(* IEC 61131-3 sources: LMM/plc/g, 5 files *)

(* ---- FB_Servo.st ---- *)
FUNCTION_BLOCK FB_Servo
(* =============================================================================
   FB_Servo — 单轴原子封装（SM3_Basic）。仅在 PRG_Axis_Control 任务内实例化。

   仲裁优先级：停止/故障 > 回零 > 绝对定位 > 相对定位 > 速度指令 > 点动。
   - 手动点动走 MC_Jog（松开即减速停）；速度指令走 MC_MoveVelocity
   - 运动切换靠 PLCopen 中止机制（新命令 FB 上升沿自动 abort 旧运动）
   - 全部运动请求撤销（松手/速度归零/停止/急停/撞限位）→ MC_Halt 减速停车
   - 硬限位：xLimEn=TRUE 时，所有模式都限制在 [rLimNeg, rLimPos] 内：
     点动/速度 越限方向被禁止；定位目标被夹紧；X 轴传 xLimEn:=FALSE
   ========================================================================== *)
VAR_IN_OUT
    Axis : AXIS_REF_SM3;
END_VAR
VAR_INPUT
    xEnable : BOOL;         (* 驱动器使能（来自 AxisCmd_xPower） *)
    xStop : BOOL;           (* 停止运动（保持使能） *)
    xResetFault : BOOL;     (* 故障复位（上升沿） *)
    xHome : BOOL;           (* 回零（电平，完成/撤销后由上层清） *)
    xMoveAbs : BOOL;        (* 绝对定位（电平保持至完成） *)
    rTargetPos : REAL;      (* 绝对目标位置 *)
    xMoveRel : BOOL;        (* 相对定位（电平保持至完成） *)
    rDist : REAL;           (* 相对距离（可正可负） *)
    xUseVelCmd : BOOL;      (* 速度指令模式（力跟随/X双驱） *)
    rVelCmd : REAL;         (* 速度给定（可正可负；|v|<1e-6 视为撤销） *)
    xJogPos : BOOL;         (* 点动+（电平，MC_Jog） *)
    xJogNeg : BOOL;         (* 点动-（电平，MC_Jog） *)
    rJogVel : REAL;         (* 点动速度（正值） *)
    rVel : REAL;            (* 定位速度（正值） *)
    rAcc : REAL;            (* 加速度 *)
    rDec : REAL;            (* 减速度 *)
    xLimEn : BOOL;          (* 硬限位使能（X=FALSE，Y/Z/R=TRUE） *)
    rLimPos : REAL;         (* 正方向硬限位（可手动改） *)
    rLimNeg : REAL;         (* 负方向硬限位（可手动改） *)
END_VAR
VAR_OUTPUT
    xPowered : BOOL;        (* 驱动器已上电 := fbPower.Status *)
    xReady : BOOL;          (* 就绪 := 上电且无故障 *)
    xMoving : BOOL;         (* 运动中（含回零） *)
    xStandstill : BOOL;     (* 静止 *)
    xHomed : BOOL;          (* 回零完成（置零后保持） *)
    xFault : BOOL;          (* 故障 := MC_ReadStatus.ErrorStop *)
    xMoveRelDone : BOOL;    (* 相对定位完成 *)
    xMoveAbsDone : BOOL;    (* 绝对定位完成 *)
    rActPos : LREAL;        (* 实际位置 *)
    (* --- 诊断输出（g 线 0.5 新增；上层可不接线，在线直接看） --- *)
    xVelReq : BOOL;         (* 诊断：仲裁后速度请求已成立 *)
    xVelBusy : BOOL;        (* 诊断：MC_MoveVelocity.Busy *)
    xVelInVel : BOOL;       (* 诊断：MC_MoveVelocity.InVelocity *)
    xErrPower : BOOL;       (* 诊断：MC_Power.Error（驱动未就绪/通讯异常） *)
    xErrVel : BOOL;         (* 诊断：MC_MoveVelocity.Error（参数/平台拒绝） *)
    xErrJog : BOOL;         (* 诊断：MC_Jog.Error *)
    xErrHalt : BOOL;        (* 诊断：MC_Halt.Error *)
    xErrHome : BOOL;        (* 诊断：MC_Home.Error *)
    xErrAbs : BOOL;         (* 诊断：MC_MoveAbsolute.Error *)
    xErrRel : BOOL;         (* 诊断：MC_MoveRelative.Error *)
END_VAR
VAR
    fbPower : MC_Power;
    fbHalt : MC_Halt;
    fbHome : MC_Home;
    fbReset : MC_Reset;
    fbReadStatus : MC_ReadStatus;
    fbReadPos : MC_ReadActualPosition;
    fbSetPos : MC_SetPosition;
    fbMoveRel : MC_MoveRelative;
    fbMoveAbs : MC_MoveAbsolute;
    fbMoveVel : MC_MoveVelocity;
    fbJog : MC_Jog;
    eDir : MC_DIRECTION;
    xReqStop : BOOL;
    xReqHome : BOOL;
    xReqAbs : BOOL;
    xReqRel : BOOL;
    xReqVel : BOOL;
    xReqJogPos : BOOL;
    xReqJogNeg : BOOL;
    xReqAny : BOOL;
    xReqHomePrev : BOOL;
    xSetZeroTrig : BOOL;
    xVelRunPrev : BOOL;
    xDirFlip : BOOL;
    xNeedStop : BOOL;
    xHaltPrev : BOOL;
    xResetPrev : BOOL;
    xBlockPos : BOOL;
    xBlockNeg : BOOL;
    rAbsTarget : REAL;
    rRelDist : REAL;
    rVelInPrev : REAL;
END_VAR

(* 1. 状态与位置 *)
fbReadStatus(Axis := Axis, Enable := TRUE);
fbReadPos(Axis := Axis, Enable := TRUE);
rActPos := fbReadPos.Position;
xStandstill := fbReadStatus.StandStill;
xFault := fbReadStatus.ErrorStop;
xMoving := fbReadStatus.DiscreteMotion OR fbReadStatus.ContinuousMotion OR fbReadStatus.Homing;

(* 2. 故障复位（上升沿） *)
fbReset(Axis := Axis, Execute := xResetFault AND NOT xResetPrev);
xResetPrev := xResetFault;

(* 3. 驱动器使能（xStop 不掉使能） *)
fbPower(Axis := Axis, Enable := TRUE,
        bRegulatorOn := xEnable AND NOT xFault,
        bDriveStart := xEnable AND NOT xFault);
xPowered := fbPower.Status;
xReady := xPowered AND NOT xFault;

(* 4. 硬限位：越限方向禁止；定位目标夹紧（已越限时仍允许向回运动） *)
xBlockPos := xLimEn AND (rActPos >= rLimPos);
xBlockNeg := xLimEn AND (rActPos <= rLimNeg);
rAbsTarget := rTargetPos;
rRelDist := rDist;
IF xLimEn THEN
    rAbsTarget := LIMIT(rLimNeg, rTargetPos, rLimPos);
    rRelDist := LIMIT(rLimNeg, rActPos + rDist, rLimPos) - rActPos;
END_IF;

(* 5. 命令仲裁：停止/故障 > 回零 > 绝对 > 相对 > 速度 > 点动 *)
xReqStop := xStop OR NOT xEnable OR xFault;
xReqHome := xHome AND NOT xReqStop;
xReqAbs := xMoveAbs AND xPowered AND NOT xReqStop AND NOT xReqHome;
xReqRel := xMoveRel AND (ABS(rRelDist) > 1.0E-9) AND xPowered
           AND NOT xReqStop AND NOT xReqHome AND NOT xReqAbs;
xReqVel := xUseVelCmd AND (ABS(rVelCmd) > 1.0E-6) AND xPowered
           AND NOT ((rVelCmd > 0.0) AND xBlockPos) AND NOT ((rVelCmd < 0.0) AND xBlockNeg)
           AND NOT xReqStop AND NOT xReqHome AND NOT xReqAbs AND NOT xReqRel;
xReqJogPos := xJogPos AND NOT xJogNeg AND NOT xBlockPos AND xPowered
              AND NOT xReqStop AND NOT xReqHome AND NOT xReqAbs AND NOT xReqRel AND NOT xReqVel;
xReqJogNeg := xJogNeg AND NOT xJogPos AND NOT xBlockNeg AND xPowered
              AND NOT xReqStop AND NOT xReqHome AND NOT xReqAbs AND NOT xReqRel AND NOT xReqVel;
xReqAny := xReqHome OR xReqAbs OR xReqRel OR xReqVel OR xReqJogPos OR xReqJogNeg;

(* 6. 回零：MC_Home(0) → MC_SetPosition(0) → xHomed *)
IF xReqHome AND NOT xReqHomePrev THEN
    xHomed := FALSE;
END_IF;
xReqHomePrev := xReqHome;
fbHome(Axis := Axis, Execute := xReqHome, Position := 0.0);
IF fbHome.Done THEN
    xSetZeroTrig := TRUE;
END_IF;
fbSetPos(Axis := Axis, Execute := xSetZeroTrig, Position := 0.0);
IF fbSetPos.Done THEN
    xHomed := TRUE;
    xSetZeroTrig := FALSE;
END_IF;

(* 7. 绝对 / 相对定位（目标已夹紧；电平保持 Execute，Done 上报） *)
fbMoveAbs(Axis := Axis, Execute := xReqAbs, Position := rAbsTarget,
          Velocity := ABS(rVel), Acceleration := rAcc, Deceleration := rDec);
fbMoveRel(Axis := Axis, Execute := xReqRel, Distance := rRelDist,
          Velocity := ABS(rVel), Acceleration := rAcc, Deceleration := rDec);
xMoveAbsDone := fbMoveAbs.Done;
xMoveRelDone := fbMoveRel.Done;

(* 8. 速度指令：MC_MoveVelocity；Velocity 取绝对值，方向走 Direction *)
(* 注意：本机 SM3 库的方向字面值是 positive/negative（非 CoDeSys 的 mcPositiveDirection） *)
IF rVelCmd >= 0.0 THEN
    eDir := positive;
ELSE
    eDir := negative;
END_IF;
(* 运行中换向：先撤 Execute 一拍，下一拍带新方向重新触发 *)
xDirFlip := xReqVel AND xVelRunPrev AND ((rVelCmd >= 0.0) <> (rVelInPrev >= 0.0));
fbMoveVel(Axis := Axis, Execute := xReqVel AND NOT xDirFlip,
          Velocity := ABS(rVelCmd), Direction := eDir,
          Acceleration := rAcc, Deceleration := rDec);
xVelRunPrev := xReqVel;
rVelInPrev := rVelCmd;

(* 9. 手动点动：MC_Jog（按住动、松开减速停；越限方向已在仲裁禁止） *)
fbJog(Axis := Axis,
      JogForward := xReqJogPos,
      JogBackward := xReqJogNeg,
      Velocity := ABS(rJogVel),
      Acceleration := rAcc,
      Deceleration := rDec);

(* 10. 停车：有使能但无任何运动请求（松手/速度归零/停止/急停/撞限位）→ MC_Halt *)
xNeedStop := xPowered AND NOT xReqAny;
fbHalt(Axis := Axis, Execute := xNeedStop AND xMoving AND NOT xHaltPrev,
       Deceleration := rDec);
xHaltPrev := xNeedStop AND xMoving;

(* 11. 诊断输出（g 线 0.5） *)
xVelReq := xReqVel;
xVelBusy := fbMoveVel.Busy;
xVelInVel := fbMoveVel.InVelocity;
xErrPower := fbPower.Error;
xErrVel := fbMoveVel.Error;
xErrJog := fbJog.Error;
xErrHalt := fbHalt.Error;
xErrHome := fbHome.Error;
xErrAbs := fbMoveAbs.Error;
xErrRel := fbMoveRel.Error;

(* ---- FB_XDual.st ---- *)
FUNCTION_BLOCK FB_XDual
(* ==============================================================================
 * FB_XDual — X 轴双驱（g 线 0.59）：单沿起步 + SM3 斜坡 + Halt 对称减速
 * 铁律：X 轴只经本 FB；FB_Servo 不得持有 X 轴实例。
 *
 *   0.44 根因：Enable 和调节器一起关 → Power FB 停转，驱动收不到卸使能；
 *   运动中切使能 + 刚上使能就 Execute → 连冲、Error 锁死第二次点动。
 *   对齐 FB_Servo：Enable 保持，bRegulatorOn/bDriveStart 跟 xRegOn；
 *   松手 Halt 脉冲刹停，双轴 standstill 后才卸调节器；2s 未静止改发 Stop。
 *   冷启动等 Status 约 80ms 且双轴 standstill 再出速度；短窗内再按不再等。
 *   0.47：禁止 300ms 超时在减速中卸使能（运动中送掉使能报错）。
 *   0.50：幅值差速不撤 Execute。必须重触发的只有换向。
 *   0.51：0.50 仍三次过冲——使能后 20ms 就 Execute（失败连打）+ 爬坡每拍改 Velocity。
 *         上使能后等 Status 80ms；Error 锁 150ms；爬坡只吃基速，到速后再跟 trim。
 *   0.52：xErrVel 不跳仍冲三次+忽快忽慢。根因是 0.51 把 xPowerSettled 绑在 standstill：
 *         轴一动就掉 Execute，松手前 Acc/Dec 反复爬。闭锁一次后保持；残差 P 降增益。
 *   0.53：xVelReq 一直 TRUE 仍冲三次。请求≠Execute；Acc=Jog 时 SM3 梯形拐点 + 使能冲击叠成三次。
 *         PLC 按用户 Acc 爬 FB 速度，SM3 Acc 抬到 ≥10 只负责跟上；松手仍 Halt。
 *   0.54：0.53 不过冲也不走。本机 Execute 保持时 Velocity 不刷新，第一拍 ~0 被锁死。
 *         上升沿一次写入目标速度 + 用户 Acc；爬坡中不改输入；到速后再跟 trim。
 *   0.55：三次过冲=Execute 被拉了三次。PRG_Logic 先清 AxisCmd 再置位，ETHERCAT(prio0)
 *         在 FALSE 空窗采到松手→Halt→再加速。第一次点动 Logic 超时约 3 拍。去抖+一次写入。
 *   0.56：偶发三次过冲。0.55 去抖保了 eMode，但 Power.Status 闪一下仍清 xStartReady，
 *         Execute 掉、锁存清 0，再启动就是又一次过冲。点动中 Execute 闭锁到松开。
 *   0.57：现场仍每次起步沿 X 往复冲 3 次（约 3s）。根因：起步=速度阶跃（Acc=25）
 *         打进 CSV 速度环，激起双驱耦合龙门 ~1Hz 纵向共振。0.53 阶梯爬速本可消过冲，
 *         但本机 Execute 保持时 Velocity 不刷新，首拍 ~0 锁死（"不过冲也不走"）。
 *   0.58：恢复 rVelSlew 阶梯爬速；爬坡期 Execute 每步重触发（OFF/ON 交替一拍，
 *         上升沿重采样）；斜率取用户 Acc/Dec 钳 [0.05, rRampAccMax]，SM3 Acc 只跟梯；
 *         松手/到位先阶梯降到 ~0 再 Halt；MoveRel 剩余≤slew²/2Dec 提前减速；
 *         到位锁 xDecelDone 禁停稳后重爬目标。
 *   0.59：0.58 每步重触发 = 250Hz 沿风暴，现场 acc=0.8 起步仍快速冲 2 次（~1s）、
 *         第三次慢、停死；M2 明显慢于 M1（两侧接受沿时刻不一致，M2 漏沿爬速落后）。
 *         改单沿起步：一个上升沿写最终目标 + 钳制用户 Acc/Dec（0.05~1.0），
 *         SM3 自带斜坡 0→目标（0.8 → 0.5s）；稳态 trim/sync 更新走限频重触发
 *         （≥200ms 一次、差值≥0.004）；减速统一 Halt（用户 Dec 对称）。
 * ============================================================================== *)
VAR_IN_OUT
    AxisM1 : AXIS_REF_SM3;
    AxisM2 : AXIS_REF_SM3;
END_VAR
VAR_INPUT
    xEnable : BOOL;
    xStop : BOOL;
    xResetFault : BOOL;
    xJogPos : BOOL;
    xJogNeg : BOOL;
    xSpinLeft : BOOL;
    xSpinRight : BOOL;
    xMoveRel : BOOL;
    rMoveDist : REAL;
    rMoveVel : REAL;
    rJogVel : REAL;
    rSpinVel : REAL;
    rHeadingErr : REAL;
    rKpTrack : REAL;
    rAcc : REAL;
    rDec : REAL;
    rTrimMax : REAL;
    xSyncEnable : BOOL := TRUE;
    rRatioM1 : REAL := 1.0;
    rRatioM2 : REAL := 1.0;
    rHeadingDeadband : REAL := 0.003;
    rTrimFilterTc : REAL := 0.05;
    rCycleSec : REAL := 0.004;
    (* 0.60 外部直控（视觉直写 M1/M2 速度）：xDirectMode=TRUE 时绕过 trim/sync *)
    xDirectMode : BOOL;
    rVelM1Direct : REAL;
    rVelM2Direct : REAL;
    tDirectRetrig : TIME := T#40MS;
END_VAR
VAR_OUTPUT
    xMoveDone : BOOL;
    rPosV : REAL;
    rSyncErr : REAL;
    rVelFactor : REAL;
    xCoupled : BOOL;
    xInGearM1 : BOOL;
    xInGearM2 : BOOL;
    xPoweredV : BOOL;
    xSyncWarn : BOOL;
    xSyncFault : BOOL;
    iState : INT;
    iHoldState : INT;
    eSlaveMode : INT;
    rVelCmdM1 : REAL;
    rVelCmdM2 : REAL;
    rPosM1 : REAL;
    rPosM2 : REAL;
    xMovingM1 : BOOL;
    xMovingM2 : BOOL;
    xStandstillM1 : BOOL;
    xStandstillM2 : BOOL;
    xPoweredM1 : BOOL;
    xPoweredM2 : BOOL;
    xReadyM1 : BOOL;
    xReadyM2 : BOOL;
    xFaultM1 : BOOL;
    xFaultM2 : BOOL;
    xVelReqM1 : BOOL;
    xVelReqM2 : BOOL;
    xVelBusyM1 : BOOL;
    xVelBusyM2 : BOOL;
    xErrPowerM1 : BOOL;
    xErrPowerM2 : BOOL;
    xErrVelM1 : BOOL;
    xErrVelM2 : BOOL;
    xVelExecM1 : BOOL;
    xVelExecM2 : BOOL;
    xVelInVelM1 : BOOL;
    xVelInVelM2 : BOOL;
    iVelExecRise : INT;
    rVelActM1Out : REAL;
    rVelActM2Out : REAL;
    xDirectActive : BOOL;
END_VAR
VAR
    fbPowerM1 : MC_Power;
    fbPowerM2 : MC_Power;
    fbResetM1 : MC_Reset;
    fbResetM2 : MC_Reset;
    fbVelM1 : MC_MoveVelocity;
    fbVelM2 : MC_MoveVelocity;
    fbHaltM1 : MC_Halt;
    fbHaltM2 : MC_Halt;
    fbStopM1 : MC_Stop;
    fbStopM2 : MC_Stop;
    eDirM1 : MC_DIRECTION;
    eDirM2 : MC_DIRECTION;
    eMode : INT;
    eModePrev : INT;
    rBase : REAL;
    rVelActM1 : REAL;
    rVelActM2 : REAL;
    rTrim : REAL;
    rTrimRaw : REAL;
    rTrimFiltered : REAL;
    rAlphaFilter : REAL;
    rUseRatioM1 : REAL;
    rUseRatioM2 : REAL;
    rSyncExpect : REAL;
    rSyncResid : REAL;
    rCorrPos : REAL;
    rCorrV1 : REAL;
    rCorrV2 : REAL;
    rVelFF1 : REAL;
    rVelFF2 : REAL;
    rKpSync : REAL := 0.05;
    rKvSync : REAL := 0.0;
    rSyncDeadband : REAL := 0.02;
    rCorrPosMax : REAL := 0.08;
    rCorrVelMax : REAL := 0.06;
    xStraightEdge : BOOL;
    xJogRaw : BOOL;
    xJogHeld : BOOL;
    tonJogOff : TON;
    tonStillM1 : TON;
    tonStillM2 : TON;
    tonHoldFallback : TON;
    tonJogGrace : TON;
    rHoldVelMax : REAL := 0.5;
    xSoftHold : BOOL;
    xSoftHoldPrev : BOOL;
    xSoftHoldLatched : BOOL;
    fbSetPosM1 : MC_SetPosition;
    fbSetPosM2 : MC_SetPosition;
    xZeroGate : BOOL;
    tonZeroDelay : TON;
    xZeroReady : BOOL;
    xZeroPulsePrev : BOOL;
    xSetPosReq : BOOL;
    xPosZeroed : BOOL;
    xErrSetPosM1 : BOOL;
    xErrSetPosM2 : BOOL;
    xResetEdge : BOOL;
    xResetPrev : BOOL;
    xDirFlipM1 : BOOL;
    xDirFlipM2 : BOOL;
    xVelRunPrevM1 : BOOL;
    xVelRunPrevM2 : BOOL;
    rVelInPrevM1 : REAL;
    rVelInPrevM2 : REAL;
    rVelAppl : REAL;
    rAccUse : REAL;
    rDecUse : REAL;
    rAccLatch : REAL;
    rDecLatch : REAL;
    rVelLatchM1 : REAL;
    rVelLatchM2 : REAL;
    xExecPrev : BOOL;
    rAccSoftMin : REAL := 0.05;
    rAccSoft : REAL;
    rDecSoft : REAL;
    rRampAccMax : REAL := 1.0;
    xDecelActive : BOOL;
    xDecelDone : BOOL;
    rDecelDist : REAL;
    xM1Decel : BOOL;
    xM2Decel : BOOL;
    xBothPowered : BOOL;
    xPowerGate : BOOL;
    xReqVelM1 : BOOL;
    xReqVelM2 : BOOL;
    xNeedHaltM1 : BOOL;
    xNeedHaltM2 : BOOL;
    xRegOn : BOOL;
    xRegOnPrev : BOOL;
    xStopping : BOOL;
    xWasStopping : BOOL;
    xHaltTrig : BOOL;
    xHaltPrev : BOOL;
    xPowerSettled : BOOL;
    xStartReady : BOOL;
    xStopFallback : BOOL;
    tonHaltWin : TON;
    tonPowerOk : TON;
    tonVelHold : TON;
    tonRampLock : TON;
    tonTrimRetrig : TON;
    xTrimWant : BOOL;
    xTrimPulse : BOOL;
    xTrimPulsePrev : BOOL;
    xMoveRelDecelTrig : BOOL;
    xExecM1 : BOOL;
    xExecHold : BOOL;
    xHaltBusy : BOOL;
    xExecBoth : BOOL;
    xDirFlipAny : BOOL;
    xVelHoldOff : BOOL;
    xErrVelPrev : BOOL;
    xRampLock : BOOL;
    rVelFbM1 : REAL;
    rVelFbM2 : REAL;
    rVelFbHoldM1 : REAL;
    rVelFbHoldM2 : REAL;
    rCorrLim : REAL;
    xMovePrev : BOOL;
    xArmed : BOOL;
    rStart : REAL;
    rAvg : REAL;
    rSyncWarnLevel : REAL := 0.05;
    rSyncFaultLevel : REAL := 0.15;
    tonSyncFault : TON;
    tonDirectRetrig : TON;
    xDirectWant : BOOL;
    xDirectPulse : BOOL;
    xDirectPulsePrev : BOOL;
    xHaltDemand : BOOL;
END_VAR

rVelFactor := 0.0;
xCoupled := FALSE;
xInGearM1 := FALSE;
xInGearM2 := FALSE;
xPoweredV := FALSE;
eSlaveMode := 0;

(* ------------------- 1. 模式 ------------------- *)
(* 点动 FALSE 短于 40ms 视为空窗，不 Halt、不撤 Execute *)
xJogRaw := (xJogPos XOR xJogNeg) OR xMoveRel;
tonJogOff(IN := xJogHeld AND NOT xJogRaw AND xEnable AND NOT xStop
           AND NOT (xSpinLeft XOR xSpinRight), PT := T#40MS);
IF xStop OR NOT xEnable THEN
    eMode := 0;
    rBase := 0.0;
    xJogHeld := FALSE;
ELSIF xSpinLeft XOR xSpinRight THEN
    IF xSpinLeft THEN
        eMode := 2;
    ELSE
        eMode := 3;
    END_IF;
    rBase := 0.0;
    xJogHeld := FALSE;
ELSIF xDirectMode THEN
    (* 0.60 外部直控优先于点动：视觉接管期间忽略点动/走距输入 *)
    eMode := 4;
    rBase := 0.0;
    xJogHeld := FALSE;
ELSIF xJogRaw THEN
    eMode := 1;
    xJogHeld := TRUE;
    IF xMoveRel THEN
        IF rMoveDist >= 0.0 THEN
            rBase := ABS(rMoveVel);
        ELSE
            rBase := -ABS(rMoveVel);
        END_IF;
    ELSIF xJogPos THEN
        rBase := ABS(rJogVel);
    ELSE
        rBase := -ABS(rJogVel);
    END_IF;
ELSIF xJogHeld AND NOT tonJogOff.Q THEN
    eMode := 1;
ELSE
    eMode := 0;
    rBase := 0.0;
    xJogHeld := FALSE;
END_IF;
iState := eMode;
xStraightEdge := (eMode = 1) AND (eModePrev <> 1);

(* ------------------- 2. 回读 + SoftHold ------------------- *)
rPosM1 := LREAL_TO_REAL(AxisM1.fActPosition);
rPosM2 := LREAL_TO_REAL(AxisM2.fActPosition);
rVelActM1 := LREAL_TO_REAL(AxisM1.fActVelocity);
rVelActM2 := LREAL_TO_REAL(AxisM2.fActVelocity);
rAvg := (rPosM1 + rPosM2) * 0.5;
rPosV := rAvg;
rSyncErr := rPosM1 - rPosM2;

xStandstillM1 := AxisM1.nAxisState = SMC_AXIS_STATE.standstill;
xStandstillM2 := AxisM2.nAxisState = SMC_AXIS_STATE.standstill;
xMovingM1 := (NOT xStandstillM1) OR (ABS(rVelActM1) > 0.01);
xMovingM2 := (NOT xStandstillM2) OR (ABS(rVelActM2) > 0.01);

tonStillM1(IN := NOT xMovingM1, PT := T#200MS);
tonStillM2(IN := NOT xMovingM2, PT := T#200MS);
tonHoldFallback(IN := (eMode = 0) AND NOT xStop AND xEnable
                    AND (ABS(rVelActM1) < rHoldVelMax) AND (ABS(rVelActM2) < rHoldVelMax),
                PT := T#2S);
IF xStop OR NOT xEnable OR (eMode <> 0) THEN
    iHoldState := 0;
    xSoftHoldLatched := FALSE;
ELSIF xSoftHoldLatched THEN
    iHoldState := 2;
ELSIF (tonStillM1.Q AND tonStillM2.Q) OR tonHoldFallback.Q THEN
    iHoldState := 2;
    xSoftHoldLatched := TRUE;
ELSE
    iHoldState := 1;
END_IF;
xSoftHold := iHoldState = 2;
xSoftHoldPrev := xSoftHold;
(* 再按起步 300ms 内隐藏 SoftHold/Halt 残留 bError，避免 Fault→StopAll 发肉 *)
tonJogGrace(IN := (eMode <> 0), PT := T#300MS);

xSyncWarn := ABS(rSyncErr) > rSyncWarnLevel;
tonSyncFault(IN := ABS(rSyncErr) > rSyncFaultLevel, PT := T#500MS);
IF tonSyncFault.Q THEN
    xSyncFault := TRUE;
END_IF;

(* ------------------- 3. 复位仅手动 ------------------- *)
fbResetM1(Axis := AxisM1, Execute := xResetFault);
fbResetM2(Axis := AxisM2, Execute := xResetFault);
IF xResetFault THEN
    xSyncFault := FALSE;
END_IF;

(* ------------------- 4. 使能：Power.Enable 常开，只切调节器 ------------------- *)
(* 松手保持调节器直到双轴 standstill。300ms 超时会在减速未完时卸使能（0.46 报错）。 *)
xWasStopping := xStopping;
IF xStop OR NOT xEnable THEN
    xStopping := FALSE;
ELSIF eMode <> 0 THEN
    xStopping := FALSE;
ELSIF xRegOnPrev THEN
    xStopping := TRUE;
END_IF;
tonHaltWin(IN := xStopping AND (eMode = 0) AND xEnable AND NOT xStop, PT := T#2S);
IF xStopping AND (eMode = 0) AND xStandstillM1 AND xStandstillM2 THEN
    xStopping := FALSE;
END_IF;
xRegOn := xEnable AND NOT xStop AND ((eMode <> 0) OR xStopping);
xStopFallback := xStopping AND tonHaltWin.Q AND NOT (xStandstillM1 AND xStandstillM2) AND NOT xDecelActive;
(* Enable 恒 TRUE，卸使能只走调节器（对齐 FB_Servo；0.44 关 Enable 导致驱动收不到） *)
fbPowerM1(Axis := AxisM1, Enable := TRUE,
          bRegulatorOn := xRegOn, bDriveStart := xRegOn);
fbPowerM2(Axis := AxisM2, Enable := TRUE,
          bRegulatorOn := xRegOn, bDriveStart := xRegOn);

xPoweredM1 := fbPowerM1.Status;
xPoweredM2 := fbPowerM2.Status;
xFaultM1 := AxisM1.bError AND xRegOn AND NOT (xSoftHold OR (iHoldState = 1) OR xStopping OR ((eMode <> 0) AND NOT tonJogGrace.Q));
xFaultM2 := AxisM2.bError AND xRegOn AND NOT (xSoftHold OR (iHoldState = 1) OR xStopping OR ((eMode <> 0) AND NOT tonJogGrace.Q));
(* 故意停调节器时仍报就绪，避免 Logic 1007 *)
xReadyM1 := xEnable AND NOT xStop AND NOT xFaultM1;
xReadyM2 := xEnable AND NOT xStop AND NOT xFaultM2;
xBothPowered := xPoweredM1 AND xPoweredM2;
xPowerGate := xEnable AND NOT xStop AND NOT xFaultM1 AND NOT xFaultM2;
tonPowerOk(IN := xRegOn AND xBothPowered AND (eMode <> 0), PT := T#80MS);
(* 冷启动闭锁一次。Status 闪烁不得清 xStartReady，否则 Execute 掉了再爬。 *)
IF (eMode = 0) OR NOT xRegOn OR xStop THEN
    xStartReady := FALSE;
ELSIF xWasStopping OR xExecHold THEN
    xStartReady := TRUE;
ELSIF tonPowerOk.Q AND xStandstillM1 AND xStandstillM2 THEN
    xStartReady := TRUE;
END_IF;
xPowerSettled := xRegOn AND (eMode <> 0) AND xStartReady
                 AND (xBothPowered OR xExecHold);

(* 置零：点动/短窗禁止；空闲自动置零会和 Halt 抢轴，只保留手动 Reset *)
IF (eMode <> 0) OR xStopping OR xStop OR NOT xEnable THEN
    xSetPosReq := FALSE;
END_IF;
xZeroGate := FALSE;
tonZeroDelay(IN := FALSE, PT := T#300MS);
xZeroReady := FALSE;
xZeroPulsePrev := FALSE;
xResetEdge := xResetFault AND NOT xResetPrev;
xResetPrev := xResetFault;
IF xResetEdge AND (eMode = 0) AND NOT xStopping THEN
    xSetPosReq := TRUE;
END_IF;
fbSetPosM1(Axis := AxisM1, Execute := xSetPosReq AND (eMode = 0) AND NOT xStopping, Position := 0.0);
fbSetPosM2(Axis := AxisM2, Execute := xSetPosReq AND (eMode = 0) AND NOT xStopping, Position := 0.0);
xErrSetPosM1 := fbSetPosM1.Error;
xErrSetPosM2 := fbSetPosM2.Error;
IF xSetPosReq THEN
    IF (fbSetPosM1.Done AND fbSetPosM2.Done) OR fbSetPosM1.Error OR fbSetPosM2.Error THEN
        xSetPosReq := FALSE;
        xPosZeroed := TRUE;
    END_IF;
END_IF;

(* ------------------- 6. 基速跟手 + 视觉差速 ------------------- *)
rAccUse := ABS(rAcc);
IF rAccUse < rAccSoftMin THEN
    rAccUse := rAccSoftMin;
END_IF;
rDecUse := ABS(rDec);
IF rDecUse < rAccSoftMin THEN
    rDecUse := rAccSoftMin;
END_IF;

(* 0.59：SM3 斜坡用钳制 Acc/Dec（0.05~rRampAccMax）。HMI 25/100 兜底不再变阶跃；
   rDecUse 保留软下限继续供 Stop 急停。 *)
rAccSoft := ABS(rAcc);
IF rAccSoft < rAccSoftMin THEN
    rAccSoft := rAccSoftMin;
END_IF;
IF rAccSoft > rRampAccMax THEN
    rAccSoft := rRampAccMax;
END_IF;
rDecSoft := ABS(rDec);
IF rDecSoft < rAccSoftMin THEN
    rDecSoft := rAccSoftMin;
END_IF;
IF rDecSoft > rRampAccMax THEN
    rDecSoft := rRampAccMax;
END_IF;

(* 0.36：禁止 PLC 再爬 rVelAppl。按下即目标速度，松开即 0，停靠 Halt。 *)
(* 0.59 注：rVelAppl 是最终目标；起步斜坡由 SM3 按 rAccSoft 生成（单沿锁存）。 *)
IF (eMode = 0) OR xStop OR NOT xEnable THEN
    rVelAppl := 0.0;
ELSIF eMode = 1 THEN
    rVelAppl := rBase;
ELSE
    rVelAppl := 0.0;
END_IF;

(* 视觉：同一条基速上 ±trim，不是第二次运动，不撤 Execute *)
rTrimRaw := 0.0;
rCorrPos := 0.0;
rCorrV1 := 0.0;
rCorrV2 := 0.0;
rUseRatioM1 := rRatioM1;
IF rUseRatioM1 < 0.1 THEN
    rUseRatioM1 := 0.1;
END_IF;
rUseRatioM2 := rRatioM2;
IF rUseRatioM2 < 0.1 THEN
    rUseRatioM2 := 0.1;
END_IF;
IF eMode = 1 THEN
    IF ABS(rHeadingErr) > ABS(rHeadingDeadband) THEN
        IF rHeadingErr > 0.0 THEN
            rTrimRaw := (rHeadingErr - ABS(rHeadingDeadband)) * rKpTrack;
        ELSE
            rTrimRaw := (rHeadingErr + ABS(rHeadingDeadband)) * rKpTrack;
        END_IF;
        rTrimRaw := LIMIT(-ABS(rTrimMax), rTrimRaw, ABS(rTrimMax));
    END_IF;
    IF rTrimFilterTc > 0.001 THEN
        rAlphaFilter := rCycleSec / (rTrimFilterTc + rCycleSec);
        rTrimFiltered := rTrimFiltered + rAlphaFilter * (rTrimRaw - rTrimFiltered);
    ELSE
        rTrimFiltered := rTrimRaw;
    END_IF;
    rTrim := rTrimFiltered;
    IF xStraightEdge THEN
        rSyncExpect := rPosM1 - rPosM2;
        rTrimFiltered := 0.0;
        rTrim := 0.0;
        xRampLock := TRUE;
    END_IF;
    rSyncExpect := rSyncExpect + (2.0 * rTrim * rCycleSec);
    rSyncResid := (rPosM1 - rPosM2) - rSyncExpect;
    rCorrLim := ABS(rCorrPosMax);
    IF ABS(rVelAppl) > 0.001 THEN
        IF (0.25 * ABS(rVelAppl)) < rCorrLim THEN
            rCorrLim := 0.25 * ABS(rVelAppl);
        END_IF;
    END_IF;
    IF xSyncEnable AND (ABS(rVelAppl) > 0.001) THEN
        IF ABS(rSyncResid) > rSyncDeadband THEN
            rCorrPos := LIMIT(-rCorrLim, rKpSync * rSyncResid, rCorrLim);
        END_IF;
        rCorrV1 := LIMIT(-ABS(rCorrVelMax), rKvSync * ((rVelAppl + rTrim) - rVelActM1), ABS(rCorrVelMax));
        rCorrV2 := LIMIT(-ABS(rCorrVelMax), rKvSync * ((rVelAppl - rTrim) - rVelActM2), ABS(rCorrVelMax));
    END_IF;
    rVelFF1 := rVelAppl + rTrim;
    rVelFF2 := rVelAppl - rTrim;
    rVelCmdM1 := (rVelFF1 - 0.5 * rCorrPos + rCorrV1) * rUseRatioM1;
    rVelCmdM2 := (rVelFF2 + 0.5 * rCorrPos + rCorrV2) * rUseRatioM2;
    IF ABS(rVelAppl) > 0.001 THEN
        IF rVelAppl > 0.0 THEN
            IF rVelCmdM1 < 0.0 THEN
                rVelCmdM1 := 0.0;
            END_IF;
            IF rVelCmdM2 < 0.0 THEN
                rVelCmdM2 := 0.0;
            END_IF;
        ELSE
            IF rVelCmdM1 > 0.0 THEN
                rVelCmdM1 := 0.0;
            END_IF;
            IF rVelCmdM2 > 0.0 THEN
                rVelCmdM2 := 0.0;
            END_IF;
        END_IF;
    END_IF;
ELSIF (eMode = 2) OR (eMode = 3) THEN
    rTrimFiltered := 0.0;
    IF eMode = 2 THEN
        rVelCmdM1 := ABS(rSpinVel) * rUseRatioM1;
    ELSE
        rVelCmdM1 := -ABS(rSpinVel) * rUseRatioM1;
    END_IF;
    rVelCmdM2 := -rVelCmdM1 * (rUseRatioM2 / rUseRatioM1);
ELSIF eMode = 4 THEN
    (* 0.60 外部直控：两个速度直接来自视觉，不做 trim/sync/斜坡 *)
    rTrimFiltered := 0.0;
    rVelCmdM1 := rVelM1Direct * rUseRatioM1;
    rVelCmdM2 := rVelM2Direct * rUseRatioM2;
ELSE
    rTrimFiltered := 0.0;
    rVelCmdM1 := rVelAppl;
    rVelCmdM2 := rVelAppl;
END_IF;
IF xStop OR NOT xEnable THEN
    rVelCmdM1 := 0.0;
    rVelCmdM2 := 0.0;
END_IF;
IF eMode <> 1 THEN
    xRampLock := FALSE;
ELSIF xRampLock THEN
    IF (ABS(rVelAppl) > 0.001)
            AND (ABS(rVelActM1) >= 0.8 * ABS(rVelAppl))
            AND (ABS(rVelActM2) >= 0.8 * ABS(rVelAppl)) THEN
        xRampLock := FALSE;
    END_IF;
END_IF;
tonRampLock(IN := xRampLock AND (eMode = 1), PT := T#800MS);
IF tonRampLock.Q THEN
    xRampLock := FALSE;
END_IF;
IF (eMode = 1) AND xRampLock THEN
    rVelFbM1 := rVelAppl * rUseRatioM1;
    rVelFbM2 := rVelAppl * rUseRatioM2;
ELSE
    rVelFbM1 := rVelCmdM1;
    rVelFbM2 := rVelCmdM2;
END_IF;
IF (eMode <> 1) OR xStraightEdge THEN
    rVelFbHoldM1 := rVelFbM1;
    rVelFbHoldM2 := rVelFbM2;
ELSE
    IF ABS(rVelFbM1 - rVelFbHoldM1) < 0.004 THEN
        rVelFbM1 := rVelFbHoldM1;
    ELSE
        rVelFbHoldM1 := rVelFbM1;
    END_IF;
    IF ABS(rVelFbM2 - rVelFbHoldM2) < 0.004 THEN
        rVelFbM2 := rVelFbHoldM2;
    ELSE
        rVelFbHoldM2 := rVelFbM2;
    END_IF;
END_IF;

(* ------------------- 7. 双轴 MoveVelocity ------------------- *)
(* 0.54：上升沿锁目标。0.58 每步重触发被 0.59 废除：250Hz 沿风暴反复踢起龙门
   1Hz 共振（现场 acc=0.8：起步快速冲 2 次 ~1s、第三次慢、停死）；两侧 FB/驱动
   接受沿时刻不一致 → M2 漏沿爬速落后（M2 明显慢）。0.59：起步只发一个上升沿，
   一次写入最终目标 + 钳制 Acc/Dec，SM3 自带斜坡 0→目标（0.8 → 0.5s）；
   稳态 trim/sync 更新走限频重触发；减速由 Halt 接管（见第 8 节）。 *)
xHaltBusy := fbHaltM1.Busy OR fbHaltM2.Busy OR fbStopM1.Busy OR fbStopM2.Busy;
IF (eMode = 1) AND xPowerGate AND xPowerSettled AND (ABS(rVelAppl) > 0.001)
        AND NOT xHaltBusy AND NOT xDecelActive AND NOT xDecelDone THEN
    xReqVelM1 := TRUE;
    xReqVelM2 := TRUE;
ELSIF ((eMode = 2) OR (eMode = 3) OR (eMode = 4)) AND xPowerGate AND xPowerSettled AND NOT xHaltBusy
        AND NOT xDecelActive AND NOT xDecelDone THEN
    IF ABS(rVelCmdM1) > 0.001 THEN
        xReqVelM1 := TRUE;
    ELSE
        xReqVelM1 := FALSE;
    END_IF;
    IF ABS(rVelCmdM2) > 0.001 THEN
        xReqVelM2 := TRUE;
    ELSE
        xReqVelM2 := FALSE;
    END_IF;
ELSE
    xReqVelM1 := FALSE;
    xReqVelM2 := FALSE;
END_IF;

xM1Decel := (NOT xReqVelM1) AND xPowerGate AND xMovingM1 AND NOT xStop AND NOT xSoftHold;
xM2Decel := (NOT xReqVelM2) AND xPowerGate AND xMovingM2 AND NOT xStop AND NOT xSoftHold;

(* 方向/换向看 FB 速度（0.54 语义）；减速期由 Halt 接管，无符号穿零 *)
IF ABS(rVelFbM1) > 0.001 THEN
    IF rVelFbM1 >= 0.0 THEN
        eDirM1 := positive;
    ELSE
        eDirM1 := negative;
    END_IF;
END_IF;
IF ABS(rVelFbM2) > 0.001 THEN
    IF rVelFbM2 >= 0.0 THEN
        eDirM2 := positive;
    ELSE
        eDirM2 := negative;
    END_IF;
END_IF;

xDirFlipM1 := xReqVelM1 AND xVelRunPrevM1
              AND (ABS(rVelFbM1) > 0.001) AND (ABS(rVelInPrevM1) > 0.001)
              AND ((rVelFbM1 >= 0.0) <> (rVelInPrevM1 >= 0.0));
xDirFlipM2 := xReqVelM2 AND xVelRunPrevM2
              AND (ABS(rVelFbM2) > 0.001) AND (ABS(rVelInPrevM2) > 0.001)
              AND ((rVelFbM2 >= 0.0) <> (rVelInPrevM2 >= 0.0));
xDirFlipAny := xDirFlipM1 OR xDirFlipM2;

IF (xErrVelM1 OR xErrVelM2) AND NOT xErrVelPrev THEN
    xVelHoldOff := TRUE;
END_IF;
tonVelHold(IN := xVelHoldOff, PT := T#150MS);
IF tonVelHold.Q THEN
    xVelHoldOff := FALSE;
END_IF;
xErrVelPrev := xErrVelM1 OR xErrVelM2;

(* 0.59 提前减速：剩余 ≤ v²/(2·Dec)，v 取双轴实际速度较大者（越保守越早触发）。
   MoveRel 未武装/静止（moved≈0）不触发，短走距不得起步即停。 *)
rDecelDist := 0.0;
IF ABS(rVelActM1) >= ABS(rVelActM2) THEN
    rDecelDist := (ABS(rVelActM1) * ABS(rVelActM1)) / (2.0 * rDecSoft);
ELSE
    rDecelDist := (ABS(rVelActM2) * ABS(rVelActM2)) / (2.0 * rDecSoft);
END_IF;
xMoveRelDecelTrig := xMoveRel AND xArmed AND (NOT xDecelDone)
                     AND (ABS(rMoveDist) > 0.001)
                     AND (ABS(rAvg - rStart) > 0.001)
                     AND (ABS(rAvg - rStart) >= ABS(rMoveDist) - rDecelDist);

(* 松手短窗 Halt 脉冲 + MoveRel 提前减速 Halt 脉冲；减速期禁重复发 *)
xHaltTrig := (xStopping AND (eMode = 0) AND NOT xStop AND NOT xStopFallback
              AND (xMovingM1 OR xMovingM2) AND NOT xDecelActive)
             OR (xMoveRelDecelTrig AND NOT xDecelActive);
(* 0.60 外部直控：任一侧目标为 0 且在动 → 双轴 Halt（停止/失联兜底由 eMode→0 处理） *)
xHaltDemand := xHaltTrig OR ((eMode = 4)
               AND (((NOT xReqVelM1) AND xMovingM1) OR ((NOT xReqVelM2) AND xMovingM2)));
xNeedHaltM1 := xHaltDemand AND NOT xHaltPrev;
xNeedHaltM2 := xNeedHaltM1;
(* 0.56 点动闭锁 + 0.59 减速期撤 Execute（Halt 接管，禁止速度指令抢轴） *)
IF xStop OR NOT xEnable THEN
    xExecHold := FALSE;
ELSIF xDecelActive THEN
    xExecHold := FALSE;
ELSIF xReqVelM1 THEN
    xExecHold := TRUE;
ELSIF (eMode = 0) OR ((eMode = 4) AND (NOT xReqVelM1 OR NOT xReqVelM2)) THEN
    xExecHold := FALSE;
END_IF;
(* 0.59 稳态 trim/sync 更新：限频重触发（≥200ms 一次）。仅非爬坡期（xRampLock 已放）、
   两侧到速、目标与锁存差 ≥0.004。脉冲期撤 Execute 一拍，下一拍上升沿重采样；
   无视觉/同步漂移时永不触发——起步到停车全程一个沿。 *)
xTrimWant := xExecHold AND (NOT xRampLock) AND xVelInVelM1 AND xVelInVelM2
             AND (NOT xDecelActive) AND (NOT xStop)
             AND ((ABS(ABS(rVelFbM1) - rVelLatchM1) >= 0.004)
                  OR (ABS(ABS(rVelFbM2) - rVelLatchM2) >= 0.004));
tonTrimRetrig(IN := xTrimWant, PT := T#200MS);
xTrimPulse := xTrimWant AND tonTrimRetrig.Q AND NOT xTrimPulsePrev;
xTrimPulsePrev := xTrimWant;
(* 0.60 外部直控：目标变化时限频重触发，跟随视觉（无变化不触发，不起沿风暴） *)
xDirectWant := (eMode = 4) AND xExecHold AND (NOT xDecelActive) AND (NOT xStop)
               AND ((ABS(ABS(rVelFbM1) - rVelLatchM1) >= 0.004)
                    OR (ABS(ABS(rVelFbM2) - rVelLatchM2) >= 0.004));
tonDirectRetrig(IN := xDirectWant, PT := tDirectRetrig);
xDirectPulse := xDirectWant AND tonDirectRetrig.Q AND NOT xDirectPulsePrev;
xDirectPulsePrev := xDirectWant;
xExecBoth := NOT xDirFlipAny AND NOT xNeedHaltM1 AND NOT xVelHoldOff AND NOT xTrimPulse
             AND NOT xDirectPulse;
xExecM1 := xExecHold AND xExecBoth;
IF xExecM1 AND NOT xExecPrev THEN
    iVelExecRise := iVelExecRise + 1;
    rVelLatchM1 := ABS(rVelFbM1);
    rVelLatchM2 := ABS(rVelFbM2);
    rAccLatch := rAccSoft;
    rDecLatch := rDecSoft;
ELSIF NOT xExecHold THEN
    rVelLatchM1 := 0.0;
    rVelLatchM2 := 0.0;
END_IF;
fbVelM1(Axis := AxisM1, Execute := xExecM1,
        Velocity := rVelLatchM1, Direction := eDirM1,
        Acceleration := rAccLatch, Deceleration := rDecLatch);
fbVelM2(Axis := AxisM2, Execute := xExecHold AND xExecBoth,
        Velocity := rVelLatchM2, Direction := eDirM2,
        Acceleration := rAccLatch, Deceleration := rDecLatch);

xExecPrev := xExecM1;
xVelRunPrevM1 := xReqVelM1;
xVelRunPrevM2 := xReqVelM2;
rVelInPrevM1 := rVelFbM1;
rVelInPrevM2 := rVelFbM2;

(* ------------------- 8. 停车 ------------------- *)
fbStopM1(Axis := AxisM1, Execute := xStop OR xStopFallback, Deceleration := rDecUse);
fbStopM2(Axis := AxisM2, Execute := xStop OR xStopFallback, Deceleration := rDecUse);
fbHaltM1(Axis := AxisM1, Execute := xNeedHaltM1, Deceleration := rDecSoft);
fbHaltM2(Axis := AxisM2, Execute := xNeedHaltM2, Deceleration := rDecSoft);
xHaltPrev := xHaltDemand;

(* ------------------- 9. 诊断与走距 ------------------- *)
xVelReqM1 := xReqVelM1;
xVelReqM2 := xReqVelM2;
xVelExecM1 := xExecM1;
xVelExecM2 := xExecHold AND xExecBoth;
xVelBusyM1 := fbVelM1.Busy;
xVelBusyM2 := fbVelM2.Busy;
xVelInVelM1 := fbVelM1.InVelocity;
xVelInVelM2 := fbVelM2.InVelocity;
xErrPowerM1 := fbPowerM1.Error;
xErrPowerM2 := fbPowerM2.Error;
xErrVelM1 := fbVelM1.Error;
xErrVelM2 := fbVelM2.Error;
(* 0.60 直控调试输出：实际速度 + 直控在役标志 *)
rVelActM1Out := rVelActM1;
rVelActM2Out := rVelActM2;
xDirectActive := (eMode = 4);

IF xStop OR NOT xEnable OR NOT xMoveRel THEN
    xArmed := FALSE;
    xMoveDone := FALSE;
ELSE
    IF xMoveRel AND NOT xMovePrev THEN
        xArmed := TRUE;
        rStart := rAvg;
    END_IF;
    xMoveDone := xArmed AND (ABS(rAvg - rStart) >= ABS(rMoveDist));
END_IF;
IF NOT xEnable THEN
    iVelExecRise := 0;
END_IF;

(* 0.59 减速状态：松手有速或 MoveRel 提前触发 → Halt 脉冲接管减速；
   双轴静止退出并置到位锁；新点动/旋转/新走距清锁。 *)
IF xMoveRel AND NOT xMovePrev THEN
    xDecelDone := FALSE;
END_IF;
IF xStop OR NOT xEnable THEN
    xDecelActive := FALSE;
    xDecelDone := FALSE;
ELSIF (eMode <> 0) AND (NOT xMoveRel) THEN
    xDecelActive := FALSE;
    xDecelDone := FALSE;
ELSIF xDecelActive THEN
    IF (NOT xMovingM1) AND (NOT xMovingM2) THEN
        xDecelActive := FALSE;
        xDecelDone := TRUE;
    END_IF;
ELSIF (eMode = 0) AND (xMovingM1 OR xMovingM2) THEN
    xDecelActive := TRUE;
ELSIF xMoveRelDecelTrig THEN
    xDecelActive := TRUE;
END_IF;
xMovePrev := xMoveRel;
eModePrev := eMode;
xRegOnPrev := xRegOn;

(* ---- PRG_Axis_Control.st ---- *)
PROGRAM PRG_Axis_Control
VAR
    fbX : FB_XDual;
    fbY : FB_Servo;
    fbZ : FB_Servo;
    fbR : FB_Servo;
    fbForce : FB_Force;
    fbFF : FB_ForceFollow;
END_VAR

(* PRG_Axis_Control — 运动独立任务(ETHERCAT 4ms)。只读 AxisCmd_*，写 AxisFb_*/rForceAct。
   禁止被其它 POU CALL；禁止写 HMI_*/报警。
   X：FB_XDual（LineTrack + 双 FB_Servo，无 Virtual/Gear）；Y/Z/R 仍 FB_Servo。 *)

(* ===== 力传感转换（本 POU 拥有 rForceAct） ===== *)
fbForce(wRaw := Force_wInRaw, rScale := Force_rScale, xEnable := Force_xEnable,
    xTare := HMI_xForceTare OR Logic_xForceTare, xUntare := HMI_xForceUntare);
Force_iRaw := fbForce.iRaw;
(* 力通讯状态由 PRG_Force485 的收发回文状态机唯一判定；
   不再用 FB_Force 的“原始值 2s 不变”看门狗覆盖，避免力稳定时误报 1005。 *)
IF NOT HMI_xForceSimEnable THEN
    rForceAct := fbForce.rForceN;
END_IF;

(* ===== X：FB_XDual（LineTrack + 双 Servo；无 Virtual/Gear） ===== *)
fbX(
    AxisM1 := Axis, AxisM2 := Axis_1,
    xEnable := AxisCmd_xPower, xStop := AxisCmd_xStopAll, xResetFault := AxisCmd_xResetFault,
    xJogPos := AxisCmd_xJogXPos, xJogNeg := AxisCmd_xJogXNeg,
    xSpinLeft := AxisCmd_xSpinLeft, xSpinRight := AxisCmd_xSpinRight,
    xMoveRel := AxisCmd_xMoveRelX, rMoveDist := AxisCmd_rMoveDistX, rMoveVel := AxisCmd_rMoveVelX,
    rJogVel := AxisCmd_rJogVelX, rSpinVel := AxisCmd_rSpinVel,
    rHeadingErr := AxisCmd_rHeadingErr, rKpTrack := AxisCmd_rTrackKp,
    rAcc := AxisCmd_rAccX, rDec := AxisCmd_rDecX,
    rTrimMax := Cfg_rPhaseMax,
    (* 0.60 视觉直控：绕过内部差速，直接给 M1/M2 速度 *)
    xDirectMode := AxisCmd_xDirectVel,
    rVelM1Direct := AxisCmd_rVelM1Set, rVelM2Direct := AxisCmd_rVelM2Set);
AxisFb_xMoveDoneX := fbX.xMoveDone;
AxisFb_rPosX := fbX.rPosV;
AxisFb_rSyncErr := fbX.rSyncErr;
AxisFb_rVelFactorX := fbX.rVelFactor;
AxisFb_xGantryCoupled := fbX.xCoupled;
AxisFb_xInGearM1 := fbX.xInGearM1;
AxisFb_xInGearM2 := fbX.xInGearM2;
AxisFb_xPoweredV := fbX.xPoweredV;
AxisFb_xSyncWarn := fbX.xSyncWarn;
AxisFb_xSyncFault := fbX.xSyncFault;
AxisFb_iGantryState := fbX.iState;
AxisFb_rVelCmdM1 := fbX.rVelCmdM1;
AxisFb_rVelCmdM2 := fbX.rVelCmdM2;
AxisFb_rPosM1 := fbX.rPosM1;
AxisFb_rPosM2 := fbX.rPosM2;
AxisFb_xMovingM1 := fbX.xMovingM1;
AxisFb_xMovingM2 := fbX.xMovingM2;
AxisFb_xStandstill1 := fbX.xStandstillM1;
AxisFb_xStandstill2 := fbX.xStandstillM2;
AxisFb_xPoweredM1 := fbX.xPoweredM1;
AxisFb_xPoweredM2 := fbX.xPoweredM2;
AxisFb_xReadyM1 := fbX.xReadyM1;
AxisFb_xReadyM2 := fbX.xReadyM2;
AxisFb_xFaultM1 := fbX.xFaultM1;
AxisFb_xFaultM2 := fbX.xFaultM2;

(* 0.60 视觉直控反馈（回给 PRG_TcpHmi 编码到状态镜像 + 视觉侧回读） *)
Direct_xActive := fbX.xDirectActive;
Direct_rVelM1Act := fbX.rVelActM1Out;
Direct_rVelM2Act := fbX.rVelActM2Out;

(* 0.63 通用双电机实际速度透传（供 PRG_TcpHmi 编码到状态 word32..38） *)
AxisFb_rVelActM1 := fbX.rVelActM1Out;
AxisFb_rVelActM2 := fbX.rVelActM2Out;

(* ===== Y：回零 > 绝对(归位) > 相对(横移) > 点动；硬限位 [Cfg_rLimYNeg, Cfg_rLimYPos] ===== *)
fbY(Axis := Axis_2, xEnable := AxisCmd_xPower, xStop := AxisCmd_xStopAll, xResetFault := AxisCmd_xResetFault,
    xHome := AxisCmd_xHomeY,
    xMoveAbs := AxisCmd_xMoveAbsY, rTargetPos := AxisCmd_rMoveAbsPosY,
    xMoveRel := AxisCmd_xMoveRelY, rDist := AxisCmd_rMoveDistY,
    xJogPos := AxisCmd_xJogYPos, xJogNeg := AxisCmd_xJogYNeg, rJogVel := AxisCmd_rJogVelY,
    rVel := AxisCmd_rMoveVelY, rAcc := AxisCmd_rAccY, rDec := AxisCmd_rDecY,
    xLimEn := TRUE, rLimPos := Cfg_rLimYPos, rLimNeg := Cfg_rLimYNeg);
AxisFb_xMoveDoneY := fbY.xMoveRelDone;

(* ===== Z：力跟随速度 > 回零 > 点动；硬限位 [Cfg_rLimZNeg, Cfg_rLimZPos] ===== *)
fbFF(rForceSet := AxisCmd_rForceSet, rForceAct := rForceAct, rKp := AxisCmd_rForceKp,
    rVelMax := AxisCmd_rForceVelMax, rDeadband := 0.5, rPosZ := fbZ.rActPos,
    rLimPos := Cfg_rLimZPos, rLimNeg := Cfg_rLimZNeg,
    xEnable := AxisCmd_xForceFollow, xInvert := FALSE);
fbZ(Axis := Axis_3, xEnable := AxisCmd_xPower, xStop := AxisCmd_xStopAll, xResetFault := AxisCmd_xResetFault,
    xHome := AxisCmd_xHomeZ,
    xUseVelCmd := AxisCmd_xForceFollow, rVelCmd := fbFF.rZVelCmd,
    xJogPos := AxisCmd_xJogZPos, xJogNeg := AxisCmd_xJogZNeg, rJogVel := AxisCmd_rJogVelZ,
    rAcc := AxisCmd_rAccZ, rDec := AxisCmd_rDecZ,
    xLimEn := TRUE, rLimPos := Cfg_rLimZPos, rLimNeg := Cfg_rLimZNeg);

(* ===== R：回零 > 保持角(绝对) > 点动；M5 门控；硬限位 [Cfg_rLimRNeg, Cfg_rLimRPos] ===== *)
fbR(Axis := Axis_4, xEnable := AxisCmd_xPower AND xM5Ready, xStop := AxisCmd_xStopAll, xResetFault := AxisCmd_xResetFault,
    xHome := AxisCmd_xHomeR,
    xMoveAbs := AxisCmd_xHoldR, rTargetPos := AxisCmd_rRHoldPos,
    xJogPos := AxisCmd_xJogRPos, xJogNeg := AxisCmd_xJogRNeg, rJogVel := AxisCmd_rJogVelR,
    rVel := AxisCmd_rJogVelR, rAcc := AxisCmd_rAccR, rDec := AxisCmd_rDecR,
    xLimEn := TRUE, rLimPos := Cfg_rLimRPos, rLimNeg := Cfg_rLimRNeg);

(* ===== Y/Z/R 反馈回写 ===== *)
AxisFb_rPosY := fbY.rActPos; AxisFb_rPosZ := fbZ.rActPos; AxisFb_rPosR := fbR.rActPos;
AxisFb_xMovingY := fbY.xMoving; AxisFb_xMovingZ := fbZ.xMoving; AxisFb_xMovingR := fbR.xMoving;
AxisFb_xStandstillY := fbY.xStandstill; AxisFb_xStandstillZ := fbZ.xStandstill; AxisFb_xStandstillR := fbR.xStandstill;
AxisFb_xPoweredY := fbY.xPowered; AxisFb_xPoweredZ := fbZ.xPowered; AxisFb_xPoweredR := fbR.xPowered;
AxisFb_xReadyY := fbY.xReady; AxisFb_xReadyZ := fbZ.xReady; AxisFb_xReadyR := fbR.xReady;
AxisFb_xHomedY := fbY.xHomed; AxisFb_xHomedZ := fbZ.xHomed; AxisFb_xHomedR := fbR.xHomed;
AxisFb_xFaultY := fbY.xFault; AxisFb_xFaultZ := fbZ.xFault; AxisFb_xFaultR := fbR.xFault;
AxisFb_xReady := AxisFb_xReadyM1 AND AxisFb_xReadyM2 AND fbY.xReady AND fbZ.xReady
    AND (NOT xM5Ready OR fbR.xReady);

(* ---- PRG_Logic.st ---- *)
PROGRAM PRG_Logic
(* PRG_Logic — 消费已仲裁 HMI_* + 面板键；写 AxisCmd_*；状态只读派生（无状态机耦合）。
   禁止 CALL Axis / FB_Servo。 *)
VAR
    tonHold : TON;
    tonReady : TON;
    xResetPulse : BOOL;
    xResetPrev : BOOL;
    xSafe : BOOL;
    xAutoStartPrev : BOOL;
    xAutoStartEdge : BOOL;
    rRHold : REAL;
    iPass : INT;
    xAutoTareSent : BOOL;
    xHomeTrigY : BOOL;
    xHomeTrigZ : BOOL;
    xHomeTrigR : BOOL;
    xHomeTrigYPrev : BOOL;
    xHomeTrigZPrev : BOOL;
    xHomeTrigRPrev : BOOL;
    xAnyHomeBusy : BOOL;
    xReadyAll : BOOL;
    xPanelSrc : BOOL;       (* eCtrlSrc=0：面板/触摸屏源 *)
    xJogXPosM : BOOL;       (* 合并后点动（HMI/Web OR 面板键） *)
    xJogXNegM : BOOL;
    xJogYPosM : BOOL;
    xJogYNegM : BOOL;
    xJogZPosM : BOOL;
    xJogZNegM : BOOL;
    xJogRPosM : BOOL;
    xJogRNegM : BOOL;
    xCmdJogXPos : BOOL;
    xCmdJogXNeg : BOOL;
    xCmdSpinL : BOOL;
    xCmdSpinR : BOOL;
    xCmdJogYPos : BOOL;
    xCmdJogYNeg : BOOL;
    xCmdJogZPos : BOOL;
    xCmdJogZNeg : BOOL;
    xCmdJogRPos : BOOL;
    xCmdJogRNeg : BOOL;
    xCmdForceFollow : BOOL;
    xCmdMoveRelX : BOOL;
    xCmdMoveRelY : BOOL;
    xCmdMoveAbsY : BOOL;
    xCmdHoldR : BOOL;
    (* 0.60 X 视觉直控仲裁 / 看门狗 *)
    tonDirectWd : TON;
    xVisSeen : BOOL;
    xVisReq : BOOL;
    xDirectSafe : BOOL;
    Vis_wSeqPrev : WORD;
    rVelM1Sel : REAL;
    rVelM2Sel : REAL;
END_VAR

(* ===== 急停锁存 / 长按复位 ===== *)
IF NOT HMI_xEStop THEN
    xEStopLatched := TRUE;
END_IF;
tonHold(IN := HMI_xStop AND HMI_xEStop, PT := T#3S);
xResetPulse := (HMI_xStopHold3s OR tonHold.Q) AND NOT xResetPrev;
xResetPrev := HMI_xStopHold3s OR tonHold.Q;
IF xResetPulse THEN
    xEStopLatched := FALSE;
    AxisCmd_xResetFault := TRUE;
    iAutoStep := 0;
    iPass := 0;
    Force_xSlaveFail := FALSE;
ELSE
    AxisCmd_xResetFault := FALSE;
END_IF;

(* 故障汇总：各轴 Errorstop（同步跳闸已废，不再 OR AxisFb_xSyncFault） *)
xFaultAggregate := AxisFb_xFaultM1 OR AxisFb_xFaultM2 OR AxisFb_xFaultY OR AxisFb_xFaultZ
    OR (xM5Ready AND AxisFb_xFaultR);

IF HMI_xAutoMode THEN eOpMode := 1; ELSE eOpMode := 0; END_IF;
HMI_eOpMode := eOpMode;

(* 安全 / 使能 —— 去耦：只看急停 + 故障 *)
xSafe := HMI_xEStop AND NOT xEStopLatched;
AxisCmd_xPower := xSafe;
AxisCmd_xStopAll := HMI_xStop OR NOT xSafe OR xFaultAggregate OR HMI_xAutoAbort;

(* ===== 0.60 X 视觉直控：Web(HMI_*) ∨ 视觉(Vis_*) 双源，视觉优先，失联即停 ===== *)
(* 视觉心跳：Vis_wSeq 变化则复位看门狗；200ms 无变化 -> 离线 *)
IF Vis_wSeq <> Vis_wSeqPrev THEN
    Vis_wSeqPrev := Vis_wSeq;
    xVisSeen := TRUE;
    tonDirectWd(IN := FALSE);
    tonDirectWd(IN := TRUE, PT := T#200MS);
END_IF;
tonDirectWd();
Direct_xOnline := xVisSeen AND NOT tonDirectWd.Q;
Direct_wSeqEcho := Vis_wSeq;

xVisReq := Vis_xEnable AND Direct_xOnline;
xDirectSafe := xSafe AND (eOpMode = 0) AND NOT HMI_xStop AND NOT xFaultAggregate;
IF xVisReq THEN
    rVelM1Sel := Vis_rVelM1Set;
    rVelM2Sel := Vis_rVelM2Set;
ELSIF HMI_xDirectEnable THEN
    rVelM1Sel := HMI_rVelM1Set;
    rVelM2Sel := HMI_rVelM2Set;
ELSE
    rVelM1Sel := 0.0;
    rVelM2Sel := 0.0;
END_IF;

Direct_xEnable := (xVisReq OR HMI_xDirectEnable) AND xDirectSafe;
AxisCmd_xDirectVel := Direct_xEnable;
AxisCmd_rVelM1Set := rVelM1Sel;
AxisCmd_rVelM2Set := rVelM2Sel;

(* 力/纠偏参数下发 *)
rForceKp := HMI_rKpForce;
IF rForceKp < 1.0E-6 THEN rForceKp := 1.0; END_IF;
AxisCmd_rForceSet := HMI_rForceSet;
AxisCmd_rForceKp := rForceKp;
AxisCmd_rForceVelMax := ABS(HMI_rAutoVelZ);
IF AxisCmd_rForceVelMax < 1.0E-6 THEN AxisCmd_rForceVelMax := ABS(HMI_rJogVelZ); END_IF;
AxisCmd_rHeadingErr := HMI_rHeadingErr;

IF HMI_xForceSimEnable THEN
    rForceAct := HMI_rForceSim;
END_IF;
HMI_rForceShow := rForceAct;

AxisCmd_rJogVelX := HMI_rJogVelX;
AxisCmd_rSpinVel := HMI_rSpinVel;
AxisCmd_rJogVelY := HMI_rJogVelY;
AxisCmd_rJogVelZ := HMI_rJogVelZ;
AxisCmd_rJogVelR := HMI_rJogVelR;
AxisCmd_rWheelBase := LIMIT(4.0, HMI_rWheelBase, 6.0);
(* 每轴加减速：仅未填(≈0)才兜底 100。X 已调到与点动速度同量级时必须原样下发。 *)
AxisCmd_rAccX := HMI_rAccX; IF AxisCmd_rAccX < 0.05 THEN AxisCmd_rAccX := 100.0; END_IF;
AxisCmd_rDecX := HMI_rDecX; IF AxisCmd_rDecX < 0.05 THEN AxisCmd_rDecX := 100.0; END_IF;
AxisCmd_rAccY := HMI_rAccY; IF AxisCmd_rAccY < 1.0 THEN AxisCmd_rAccY := 100.0; END_IF;
AxisCmd_rDecY := HMI_rDecY; IF AxisCmd_rDecY < 1.0 THEN AxisCmd_rDecY := 100.0; END_IF;
AxisCmd_rAccZ := HMI_rAccZ; IF AxisCmd_rAccZ < 1.0 THEN AxisCmd_rAccZ := 100.0; END_IF;
AxisCmd_rDecZ := HMI_rDecZ; IF AxisCmd_rDecZ < 1.0 THEN AxisCmd_rDecZ := 100.0; END_IF;
AxisCmd_rAccR := HMI_rAccR; IF AxisCmd_rAccR < 1.0 THEN AxisCmd_rAccR := 100.0; END_IF;
AxisCmd_rDecR := HMI_rDecR; IF AxisCmd_rDecR < 1.0 THEN AxisCmd_rDecR := 100.0; END_IF;

(* 限位联锁：物理限位输入 ∨ 可配置硬限位（Cfg_rLim*，FB_Servo 内另有最终闸门） *)
xIlk_BlockYPlus := I_xLimYPos OR (AxisFb_rPosY >= Cfg_rLimYPos);
xIlk_BlockYNeg := I_xLimYNeg OR (AxisFb_rPosY <= Cfg_rLimYNeg);
xIlk_BlockZPlus := I_xLimZPos OR (AxisFb_rPosZ >= Cfg_rLimZPos);
xIlk_BlockZNeg := I_xLimZNeg OR (AxisFb_rPosZ <= Cfg_rLimZNeg);

(* 运动位先写入局部，扫描结束一次性交给 AxisCmd。
   禁止先清 GVL 再置位：ETHERCAT 优先级更高，会采到 FALSE 空窗，点动 Acc 被重爬三次。 *)
xCmdJogXPos := FALSE; xCmdJogXNeg := FALSE;
xCmdSpinL := FALSE; xCmdSpinR := FALSE;
xCmdJogYPos := FALSE; xCmdJogYNeg := FALSE;
xCmdJogZPos := FALSE; xCmdJogZNeg := FALSE;
xCmdJogRPos := FALSE; xCmdJogRNeg := FALSE;
xCmdForceFollow := FALSE;
xCmdMoveRelX := FALSE;
xCmdMoveRelY := FALSE;
xCmdMoveAbsY := FALSE;
xCmdHoldR := FALSE;
(* 视觉差速：手动点动与自动走距都下发 Kp；FB 仅在直行模式用 *)
AxisCmd_rTrackKp := HMI_rKpTrack;
Logic_xForceTare := FALSE;

xAutoStartEdge := HMI_xAutoStart AND NOT xAutoStartPrev;
xAutoStartPrev := HMI_xAutoStart;

IF HMI_xAutoAbort OR NOT xSafe OR xFaultAggregate THEN
    iAutoStep := 0;
    iPass := 0;
    HMI_xAutoBusy := FALSE;
END_IF;

(* ===== 点动源合并：面板键（仅面板/触摸屏源时）OR 触摸屏/Web ===== *)
xPanelSrc := (eCtrlSrc = 0);
xJogXPosM := HMI_xJogXPos OR (xPanelSrc AND JogFwd);
xJogXNegM := HMI_xJogXNeg OR (xPanelSrc AND JogBwd);
xJogYPosM := HMI_xJogYPos OR (xPanelSrc AND JogRight);
xJogYNegM := HMI_xJogYNeg OR (xPanelSrc AND JogLeft);
xJogZPosM := HMI_xJogZPos OR (xPanelSrc AND JogUp);
xJogZNegM := HMI_xJogZNeg OR (xPanelSrc AND JogDown);
xJogRPosM := HMI_xJogRPos OR (xPanelSrc AND JogClockAdd);
xJogRNegM := HMI_xJogRNeg OR (xPanelSrc AND JogClockMis);

(* ===== 手动 ===== *)
IF xSafe AND (eOpMode = 0) AND NOT HMI_xStop AND NOT xFaultAggregate THEN
    (* 直控在役时屏蔽 X 手动（旋转/点动），速度由视觉/Web 直控通道给 *)
    IF (HMI_xSpinLeft XOR HMI_xSpinRight) AND NOT Direct_xEnable THEN
        xCmdSpinL := HMI_xSpinLeft;
        xCmdSpinR := HMI_xSpinRight;
    ELSIF (xJogXPosM XOR xJogXNegM) AND NOT Direct_xEnable THEN
        xCmdJogXPos := xJogXPosM;
        xCmdJogXNeg := xJogXNegM;
    END_IF;
    xCmdJogYPos := xJogYPosM AND NOT xIlk_BlockYPlus;
    xCmdJogYNeg := xJogYNegM AND NOT xIlk_BlockYNeg;
    IF HMI_xForceGuide THEN
        xCmdForceFollow := TRUE;
    ELSE
        xCmdJogZPos := xJogZPosM AND NOT xIlk_BlockZPlus;
        xCmdJogZNeg := xJogZNegM AND NOT xIlk_BlockZNeg;
    END_IF;
    IF xM5Ready THEN
        xCmdJogRPos := xJogRPosM;
        xCmdJogRNeg := xJogRNegM;
    END_IF;
END_IF;

(* ===== 自动多道循环 ===== *)
IF xSafe AND (eOpMode = 1) AND NOT HMI_xStop AND NOT xFaultAggregate THEN
    IF iAutoStep = 0 AND xAutoStartEdge THEN
        rRHold := AxisFb_rPosR;
        xAutoTareSent := FALSE;
        HMI_xAutoDone := FALSE;
        HMI_xAutoBusy := TRUE;
        iPass := 1;
        iAutoStep := 1;
    END_IF;

    CASE iAutoStep OF
        1:
            xCmdHoldR := TRUE;
            AxisCmd_rRHoldPos := rRHold;
            AxisCmd_rTrackKp := HMI_rKpTrack;
            AxisCmd_rMoveDistX := HMI_rAutoDistX;
            AxisCmd_rMoveVelX := HMI_rAutoVelX;
            xCmdMoveRelX := TRUE;
            IF AxisFb_xMoveDoneX THEN
                xCmdMoveRelX := FALSE;
                iAutoStep := 2;
            END_IF;
        2:
            xCmdHoldR := TRUE;
            AxisCmd_rRHoldPos := rRHold;
            AxisCmd_rMoveAbsPosY := 0.0;
            AxisCmd_rMoveVelY := HMI_rAutoVelY;
            xCmdMoveAbsY := TRUE;
            IF AxisFb_xStandstillY AND (ABS(AxisFb_rPosY) < 0.005) THEN
                xCmdMoveAbsY := FALSE;
                xAutoTareSent := FALSE;
                iAutoStep := 3;
            END_IF;
        3:
            xCmdHoldR := TRUE;
            AxisCmd_rRHoldPos := rRHold;
            IF NOT xAutoTareSent THEN
                Logic_xForceTare := TRUE;
                xAutoTareSent := TRUE;
            END_IF;
            xCmdForceFollow := TRUE;
            IF rForceAct >= HMI_rForceSet THEN
                iAutoStep := 4;
            END_IF;
        4:
            xCmdHoldR := TRUE;
            AxisCmd_rRHoldPos := rRHold;
            xCmdForceFollow := TRUE;
            AxisCmd_rMoveDistY := AxisCmd_rWheelBase;
            AxisCmd_rMoveVelY := HMI_rAutoVelY;
            xCmdMoveRelY := TRUE;
            IF AxisFb_xMoveDoneY THEN
                xCmdMoveRelY := FALSE;
                iAutoStep := 5;
            END_IF;
        5:
            IF iPass < HMI_iAutoPasses THEN
                iPass := iPass + 1;
                iAutoStep := 1;
            ELSE
                iAutoStep := 6;
            END_IF;
        6:
            HMI_xAutoBusy := FALSE;
            HMI_xAutoDone := TRUE;
            iAutoStep := 0;
            iPass := 0;
    END_CASE;
END_IF;

(* ===== 回零：Y/Z/R；同时只回一轴 ===== *)
xHomeTrigY := HMI_xHomeY OR ((HMI_iHomeAxis = 1) AND HMI_xHomeExec);
xHomeTrigZ := HMI_xHomeZ OR ((HMI_iHomeAxis = 2) AND HMI_xHomeExec);
xHomeTrigR := HMI_xHomeR OR ((HMI_iHomeAxis = 3) AND HMI_xHomeExec);
xAnyHomeBusy := AxisCmd_xHomeY OR AxisCmd_xHomeZ OR AxisCmd_xHomeR;

IF AxisCmd_xStopAll OR NOT xSafe OR xFaultAggregate THEN
    AxisCmd_xHomeY := FALSE;
    AxisCmd_xHomeZ := FALSE;
    AxisCmd_xHomeR := FALSE;
ELSE
    IF AxisCmd_xHomeY AND AxisFb_xHomedY THEN AxisCmd_xHomeY := FALSE; END_IF;
    IF AxisCmd_xHomeZ AND AxisFb_xHomedZ THEN AxisCmd_xHomeZ := FALSE; END_IF;
    IF AxisCmd_xHomeR AND AxisFb_xHomedR THEN AxisCmd_xHomeR := FALSE; END_IF;
    IF (eOpMode = 0) AND NOT HMI_xStop THEN
        IF xHomeTrigY AND NOT xHomeTrigYPrev AND NOT xAnyHomeBusy THEN
            AxisCmd_xHomeY := TRUE;
        ELSIF xHomeTrigZ AND NOT xHomeTrigZPrev AND NOT xAnyHomeBusy THEN
            AxisCmd_xHomeZ := TRUE;
        ELSIF xHomeTrigR AND NOT xHomeTrigRPrev AND NOT xAnyHomeBusy AND xM5Ready THEN
            AxisCmd_xHomeR := TRUE;
        END_IF;
    END_IF;
END_IF;
xHomeTrigYPrev := xHomeTrigY;
xHomeTrigZPrev := xHomeTrigZ;
xHomeTrigRPrev := xHomeTrigR;

IF AxisCmd_xHomeY THEN xCmdJogYPos := FALSE; xCmdJogYNeg := FALSE; END_IF;
IF AxisCmd_xHomeZ THEN xCmdJogZPos := FALSE; xCmdJogZNeg := FALSE; xCmdForceFollow := FALSE; END_IF;
IF AxisCmd_xHomeR THEN xCmdJogRPos := FALSE; xCmdJogRNeg := FALSE; END_IF;

(* 本扫描只写一次 GVL，ETHERCAT 不会采到中途 FALSE *)
AxisCmd_xJogXPos := xCmdJogXPos; AxisCmd_xJogXNeg := xCmdJogXNeg;
AxisCmd_xSpinLeft := xCmdSpinL; AxisCmd_xSpinRight := xCmdSpinR;
AxisCmd_xJogYPos := xCmdJogYPos; AxisCmd_xJogYNeg := xCmdJogYNeg;
AxisCmd_xJogZPos := xCmdJogZPos; AxisCmd_xJogZNeg := xCmdJogZNeg;
AxisCmd_xJogRPos := xCmdJogRPos; AxisCmd_xJogRNeg := xCmdJogRNeg;
AxisCmd_xForceFollow := xCmdForceFollow;
AxisCmd_xMoveRelX := xCmdMoveRelX;
AxisCmd_xMoveRelY := xCmdMoveRelY;
AxisCmd_xMoveAbsY := xCmdMoveAbsY;
AxisCmd_xHoldR := xCmdHoldR;

HMI_xHomedY := AxisFb_xHomedY;
HMI_xHomedZ := AxisFb_xHomedZ;
HMI_xHomedR := AxisFb_xHomedR;
HMI_xHomeBusyY := AxisCmd_xHomeY;
HMI_xHomeBusyZ := AxisCmd_xHomeZ;
HMI_xHomeBusyR := AxisCmd_xHomeR;

(* 使能就绪诊断 → 1007 *)
xReadyAll := AxisFb_xReadyM1 AND AxisFb_xReadyM2 AND AxisFb_xReadyY AND AxisFb_xReadyZ
    AND (NOT xM5Ready OR AxisFb_xReadyR);
tonReady(IN := AxisCmd_xPower AND NOT xReadyAll AND NOT xFaultAggregate, PT := T#2S);

(* 报警 *)
IF xEStopLatched OR NOT HMI_xEStop THEN
    iAlarmID := 1001;
ELSIF AxisFb_xFaultM1 OR AxisFb_xFaultM2 OR AxisFb_xFaultY OR AxisFb_xFaultZ
        OR (xM5Ready AND AxisFb_xFaultR) THEN
    iAlarmID := 1002;
ELSIF tonReady.Q THEN
    iAlarmID := 1007;
ELSIF NOT HMI_xForceSimEnable AND Force_xSlaveFail THEN
    iAlarmID := 1006;
ELSIF NOT HMI_xForceSimEnable AND Force_xTimeout THEN
    iAlarmID := 1005;
ELSE
    iAlarmID := 0;
END_IF;

(* 状态灯（只读派生，不互锁） *)
Dev_xError := xFaultAggregate;
Dev_xRun := xSafe AND NOT HMI_xStop AND NOT xFaultAggregate;
Dev_xStop := NOT Dev_xRun AND NOT Dev_xError;
HMI_xDevError := Dev_xError;
HMI_xDevRun := Dev_xRun;
HMI_xDevStop := Dev_xStop;
IF Dev_xError THEN HMI_eDevState := 2;
ELSIF Dev_xRun THEN HMI_eDevState := 1;
ELSE HMI_eDevState := 0; END_IF;

HMI_iAutoStepShow := iAutoStep;
HMI_xLampEStop := xEStopLatched OR NOT HMI_xEStop;
HMI_xLampEnableOk := Dev_xRun;
HMI_xLampFault := xFaultAggregate;
HMI_iAlarmShow := iAlarmID;

StopLamp := Dev_xStop;
StartLamp := Dev_xRun;

(* ---- PRG_TcpHmi.st ---- *)
PROGRAM PRG_TcpHmi
(* PRG_TcpHmi — Modbus TCP 过程映像编解码 + 控制源仲裁。
   PLC=从站；Gateway=主站：FC16 写 Holding1000 命令 / FC03 读 Holding1100 状态。
   eCtrlSrc 为 GVL 变量：0=面板/触摸屏 1=远程(Web)。
   0.68：镜像 96 字；命令 word60..75 全轴直控；状态 word39..45 回传。
   0.70：命令 word5 bit11 力峰值复位；状态 word46/47 力峰值 ×100、word48 力原始计数。 *)
SM3001:=TRUE;
VAR
    xInit : BOOL;
    xPanelOp : BOOL;
    xTcpOp : BOOL;
    xValid : BOOL;
    wMagic : WORD;
    wVersion : WORD;
    wSeqHead : WORD;
    wSeqTail : WORD;
    wHeartbeat : WORD;
    dwTmp : DWORD;
    diTmp : DINT;
    iTmp : INT;
    i : INT;
    tonHb : TON;
END_VAR

(* PRG_TcpHmi — Modbus TCP 过程映像编解码 + 控制源仲裁。
   PLC=Master 读 Holding1000 / 写 Holding1100；Gateway=Server。
   eCtrlSrc 为 GVL 变量：0=面板/触摸屏 1=远程(Web)。 *)

IF NOT xInit THEN
    Tcp_xEStop := TRUE;
    Tcp_rJogVelX := 0.4; Tcp_rSpinVel := 0.3;
    Tcp_rJogVelY := 0.3; Tcp_rJogVelZ := 0.2; Tcp_rJogVelR := 0.2;
    Tcp_rAutoDistX := 1.0; Tcp_rAutoVelX := 0.4;
    Tcp_rAutoVelY := 0.3; Tcp_rAutoVelZ := 0.15;
    Tcp_rWheelBase := 5.0; Tcp_rForceSet := 100.0;
    Tcp_xForceSimEnable := FALSE;
    Tcp_iAutoPasses := 1;
    Tcp_rHeadingErr := 0.0;
    Tcp_rKpTrack := 0.0; Tcp_rKpForce := 1.0;
    Tcp_rAccX := 100.0; Tcp_rDecX := 100.0;
    Tcp_rAccY := 100.0; Tcp_rDecY := 100.0;
    Tcp_rAccZ := 100.0; Tcp_rDecZ := 100.0;
    Tcp_rAccR := 100.0; Tcp_rDecR := 100.0;
    Tcp_iCommStatus := 0;
    Tcp_wLastHb := 0; Tcp_wLastSeq := 16#FFFF; Tcp_wStatusSeq := 0;
    Tcp_iDirectModeX := 0; Tcp_iDirectModeY := 0; Tcp_iDirectModeZ := 0; Tcp_iDirectModeR := 0;
    Tcp_rDirectPosX := 0.0; Tcp_rDirectVelY := 0.0; Tcp_rDirectPosY := 0.0;
    Tcp_rDirectVelZ := 0.0; Tcp_rDirectPosZ := 0.0; Tcp_rDirectVelR := 0.0; Tcp_rDirectPosR := 0.0;
    Tcp_wDirectSeq := 0;
    tonHb(IN := FALSE);
    xInit := TRUE;
END_IF;

(* ===== 命令快照解码 ===== *)
wMagic := MB_CmdIn[0];
wVersion := MB_CmdIn[1];
wSeqHead := MB_CmdIn[2];
wHeartbeat := MB_CmdIn[3];
wSeqTail := MB_CmdIn[95];
xValid := (wMagic = 19533) AND (wVersion = 256) AND (wSeqHead = wSeqTail);
IF xValid THEN
    Tcp_iCommStatus := 1;
    IF wHeartbeat <> Tcp_wLastHb THEN
        tonHb(IN := FALSE);
        tonHb(IN := TRUE, PT := T#1S);
        Tcp_wLastHb := wHeartbeat;
    END_IF;
    IF wSeqHead <> Tcp_wLastSeq THEN
        Tcp_wLastSeq := wSeqHead;
        Tcp_xEStop := (MB_CmdIn[4] AND 1) <> 0;
        Tcp_xStop := (MB_CmdIn[4] AND 2) <> 0;
        Tcp_xStopHold3s := (MB_CmdIn[4] AND 4) <> 0;
        Tcp_xStart := (MB_CmdIn[4] AND 8) <> 0;
        Tcp_xEnable := (MB_CmdIn[4] AND 16) <> 0;
        Tcp_xAutoMode := (MB_CmdIn[4] AND 32) <> 0;
        Tcp_xJogXPos := (MB_CmdIn[4] AND 64) <> 0;
        Tcp_xJogXNeg := (MB_CmdIn[4] AND 128) <> 0;
        Tcp_xSpinLeft := (MB_CmdIn[4] AND 256) <> 0;
        Tcp_xSpinRight := (MB_CmdIn[4] AND 512) <> 0;
        Tcp_xJogYPos := (MB_CmdIn[4] AND 1024) <> 0;
        Tcp_xJogYNeg := (MB_CmdIn[4] AND 2048) <> 0;
        Tcp_xJogZPos := (MB_CmdIn[4] AND 4096) <> 0;
        Tcp_xJogZNeg := (MB_CmdIn[4] AND 8192) <> 0;
        Tcp_xJogRPos := (MB_CmdIn[4] AND 16384) <> 0;
        Tcp_xJogRNeg := (MB_CmdIn[4] AND 32768) <> 0;
        Tcp_xHomeY := (MB_CmdIn[5] AND 1) <> 0;
        Tcp_xHomeZ := (MB_CmdIn[5] AND 2) <> 0;
        Tcp_xHomeR := (MB_CmdIn[5] AND 4) <> 0;
        Tcp_xHomeExec := (MB_CmdIn[5] AND 8) <> 0;
        Tcp_xAutoStart := (MB_CmdIn[5] AND 16) <> 0;
        Tcp_xAutoAbort := (MB_CmdIn[5] AND 32) <> 0;
        Tcp_xForceSimEnable := (MB_CmdIn[5] AND 64) <> 0;
        Tcp_xForceTare := (MB_CmdIn[5] AND 128) <> 0;
        Tcp_xForceUntare := (MB_CmdIn[5] AND 256) <> 0;
        Tcp_xForceGuide := (MB_CmdIn[5] AND 512) <> 0;
        Tcp_xForcePeakReset := (MB_CmdIn[5] AND 2048) <> 0;
        (* 0.60 X 直控：Web 通道 word5 bit10 + word54/55；视觉块 word56..59 每周期直读 *)
        HMI_xDirectEnable := (MB_CmdIn[5] AND 1024) <> 0;
        HMI_rVelM1Set := INT_TO_REAL(WORD_TO_INT(MB_CmdIn[54])) / 1000.0;
        HMI_rVelM2Set := INT_TO_REAL(WORD_TO_INT(MB_CmdIn[55])) / 1000.0;
        Vis_xEnable := (MB_CmdIn[56] AND 1) <> 0;
        Vis_wSeq := MB_CmdIn[57];
        Vis_rVelM1Set := INT_TO_REAL(WORD_TO_INT(MB_CmdIn[58])) / 1000.0;
        Vis_rVelM2Set := INT_TO_REAL(WORD_TO_INT(MB_CmdIn[59])) / 1000.0;
        Tcp_iHomeAxis := WORD_TO_INT(MB_CmdIn[6]);
        Tcp_iAutoPasses := WORD_TO_INT(MB_CmdIn[7]);
        dwTmp := SHL(WORD_TO_DWORD(MB_CmdIn[8]), 16) OR WORD_TO_DWORD(MB_CmdIn[9]);
        Tcp_rJogVelX := DINT_TO_REAL(DWORD_TO_DINT(dwTmp)) / 1000.0;
        dwTmp := SHL(WORD_TO_DWORD(MB_CmdIn[10]), 16) OR WORD_TO_DWORD(MB_CmdIn[11]);
        Tcp_rSpinVel := DINT_TO_REAL(DWORD_TO_DINT(dwTmp)) / 1000.0;
        dwTmp := SHL(WORD_TO_DWORD(MB_CmdIn[12]), 16) OR WORD_TO_DWORD(MB_CmdIn[13]);
        Tcp_rJogVelY := DINT_TO_REAL(DWORD_TO_DINT(dwTmp)) / 1000.0;
        dwTmp := SHL(WORD_TO_DWORD(MB_CmdIn[14]), 16) OR WORD_TO_DWORD(MB_CmdIn[15]);
        Tcp_rJogVelZ := DINT_TO_REAL(DWORD_TO_DINT(dwTmp)) / 1000.0;
        dwTmp := SHL(WORD_TO_DWORD(MB_CmdIn[16]), 16) OR WORD_TO_DWORD(MB_CmdIn[17]);
        Tcp_rJogVelR := DINT_TO_REAL(DWORD_TO_DINT(dwTmp)) / 1000.0;
        dwTmp := SHL(WORD_TO_DWORD(MB_CmdIn[18]), 16) OR WORD_TO_DWORD(MB_CmdIn[19]);
        Tcp_rAutoDistX := DINT_TO_REAL(DWORD_TO_DINT(dwTmp)) / 1000.0;
        dwTmp := SHL(WORD_TO_DWORD(MB_CmdIn[20]), 16) OR WORD_TO_DWORD(MB_CmdIn[21]);
        Tcp_rAutoVelX := DINT_TO_REAL(DWORD_TO_DINT(dwTmp)) / 1000.0;
        dwTmp := SHL(WORD_TO_DWORD(MB_CmdIn[22]), 16) OR WORD_TO_DWORD(MB_CmdIn[23]);
        Tcp_rAutoVelY := DINT_TO_REAL(DWORD_TO_DINT(dwTmp)) / 1000.0;
        dwTmp := SHL(WORD_TO_DWORD(MB_CmdIn[24]), 16) OR WORD_TO_DWORD(MB_CmdIn[25]);
        Tcp_rAutoVelZ := DINT_TO_REAL(DWORD_TO_DINT(dwTmp)) / 1000.0;
        dwTmp := SHL(WORD_TO_DWORD(MB_CmdIn[26]), 16) OR WORD_TO_DWORD(MB_CmdIn[27]);
        Tcp_rWheelBase := DINT_TO_REAL(DWORD_TO_DINT(dwTmp)) / 1000.0;
        dwTmp := SHL(WORD_TO_DWORD(MB_CmdIn[28]), 16) OR WORD_TO_DWORD(MB_CmdIn[29]);
        Tcp_rForceSet := DINT_TO_REAL(DWORD_TO_DINT(dwTmp)) / 100.0;
        dwTmp := SHL(WORD_TO_DWORD(MB_CmdIn[30]), 16) OR WORD_TO_DWORD(MB_CmdIn[31]);
        Tcp_rForceSim := DINT_TO_REAL(DWORD_TO_DINT(dwTmp)) / 100.0;
        dwTmp := SHL(WORD_TO_DWORD(MB_CmdIn[32]), 16) OR WORD_TO_DWORD(MB_CmdIn[33]);
        Tcp_rHeadingErr := DINT_TO_REAL(DWORD_TO_DINT(dwTmp)) / 1000.0;
        dwTmp := SHL(WORD_TO_DWORD(MB_CmdIn[34]), 16) OR WORD_TO_DWORD(MB_CmdIn[35]);
        Tcp_rKpTrack := DINT_TO_REAL(DWORD_TO_DINT(dwTmp)) / 1000.0;
        dwTmp := SHL(WORD_TO_DWORD(MB_CmdIn[36]), 16) OR WORD_TO_DWORD(MB_CmdIn[37]);
        Tcp_rKpForce := DINT_TO_REAL(DWORD_TO_DINT(dwTmp)) / 1000.0;
        dwTmp := SHL(WORD_TO_DWORD(MB_CmdIn[38]), 16) OR WORD_TO_DWORD(MB_CmdIn[39]);
        Tcp_rAccX := DINT_TO_REAL(DWORD_TO_DINT(dwTmp)) / 1000.0;
        dwTmp := SHL(WORD_TO_DWORD(MB_CmdIn[40]), 16) OR WORD_TO_DWORD(MB_CmdIn[41]);
        Tcp_rDecX := DINT_TO_REAL(DWORD_TO_DINT(dwTmp)) / 1000.0;
        dwTmp := SHL(WORD_TO_DWORD(MB_CmdIn[42]), 16) OR WORD_TO_DWORD(MB_CmdIn[43]);
        Tcp_rAccY := DINT_TO_REAL(DWORD_TO_DINT(dwTmp)) / 1000.0;
        dwTmp := SHL(WORD_TO_DWORD(MB_CmdIn[44]), 16) OR WORD_TO_DWORD(MB_CmdIn[45]);
        Tcp_rDecY := DINT_TO_REAL(DWORD_TO_DINT(dwTmp)) / 1000.0;
        dwTmp := SHL(WORD_TO_DWORD(MB_CmdIn[46]), 16) OR WORD_TO_DWORD(MB_CmdIn[47]);
        Tcp_rAccZ := DINT_TO_REAL(DWORD_TO_DINT(dwTmp)) / 1000.0;
        dwTmp := SHL(WORD_TO_DWORD(MB_CmdIn[48]), 16) OR WORD_TO_DWORD(MB_CmdIn[49]);
        Tcp_rDecZ := DINT_TO_REAL(DWORD_TO_DINT(dwTmp)) / 1000.0;
        dwTmp := SHL(WORD_TO_DWORD(MB_CmdIn[50]), 16) OR WORD_TO_DWORD(MB_CmdIn[51]);
        Tcp_rAccR := DINT_TO_REAL(DWORD_TO_DINT(dwTmp)) / 1000.0;
        dwTmp := SHL(WORD_TO_DWORD(MB_CmdIn[52]), 16) OR WORD_TO_DWORD(MB_CmdIn[53]);
        Tcp_rDecR := DINT_TO_REAL(DWORD_TO_DINT(dwTmp)) / 1000.0;
        (* 0.68 全轴直控命令 word60..75；视觉与操作员共用同一镜像 *)
        (* 模式字 word60/63/67/71：用局部索引读取（word63 与旧 tailSequence 同号，静态规则勿再出现直写下标） *)
        i := 60; iTmp := WORD_TO_INT(MB_CmdIn[i]); Tcp_iDirectModeX := INT_TO_UINT(iTmp);
        dwTmp := SHL(WORD_TO_DWORD(MB_CmdIn[61]), 16) OR WORD_TO_DWORD(MB_CmdIn[62]);
        Tcp_rDirectPosX := DINT_TO_REAL(DWORD_TO_DINT(dwTmp)) / 1000.0;
        i := 63; iTmp := WORD_TO_INT(MB_CmdIn[i]); Tcp_iDirectModeY := INT_TO_UINT(iTmp);
        Tcp_rDirectVelY := INT_TO_REAL(WORD_TO_INT(MB_CmdIn[64])) / 1000.0;
        dwTmp := SHL(WORD_TO_DWORD(MB_CmdIn[65]), 16) OR WORD_TO_DWORD(MB_CmdIn[66]);
        Tcp_rDirectPosY := DINT_TO_REAL(DWORD_TO_DINT(dwTmp)) / 1000.0;
        i := 67; iTmp := WORD_TO_INT(MB_CmdIn[i]); Tcp_iDirectModeZ := INT_TO_UINT(iTmp);
        Tcp_rDirectVelZ := INT_TO_REAL(WORD_TO_INT(MB_CmdIn[68])) / 1000.0;
        dwTmp := SHL(WORD_TO_DWORD(MB_CmdIn[69]), 16) OR WORD_TO_DWORD(MB_CmdIn[70]);
        Tcp_rDirectPosZ := DINT_TO_REAL(DWORD_TO_DINT(dwTmp)) / 1000.0;
        i := 71; iTmp := WORD_TO_INT(MB_CmdIn[i]); Tcp_iDirectModeR := INT_TO_UINT(iTmp);
        Tcp_rDirectVelR := INT_TO_REAL(WORD_TO_INT(MB_CmdIn[72])) / 1000.0;
        dwTmp := SHL(WORD_TO_DWORD(MB_CmdIn[73]), 16) OR WORD_TO_DWORD(MB_CmdIn[74]);
        Tcp_rDirectPosR := DINT_TO_REAL(DWORD_TO_DINT(dwTmp)) / 1000.0;
        Tcp_wDirectSeq := MB_CmdIn[75];
    END_IF;
ELSIF wMagic <> 0 AND wMagic <> 19533 THEN
    Tcp_iCommStatus := 2;
ELSIF wSeqHead <> wSeqTail THEN
    Tcp_iCommStatus := 3;
END_IF;

(* 0.68 直控命令影子 → HMI_*：每周期跟随；心跳由 PRG_Logic 看门狗判定 *)
HMI_iDirectModeX := Tcp_iDirectModeX;
HMI_rDirectPosX := Tcp_rDirectPosX;
HMI_iDirectModeY := Tcp_iDirectModeY;
HMI_rDirectVelY := Tcp_rDirectVelY;
HMI_rDirectPosY := Tcp_rDirectPosY;
HMI_iDirectModeZ := Tcp_iDirectModeZ;
HMI_rDirectVelZ := Tcp_rDirectVelZ;
HMI_rDirectPosZ := Tcp_rDirectPosZ;
HMI_iDirectModeR := Tcp_iDirectModeR;
HMI_rDirectVelR := Tcp_rDirectVelR;
HMI_rDirectPosR := Tcp_rDirectPosR;
HMI_wDirectSeq := Tcp_wDirectSeq;

tonHb();
IF tonHb.Q OR Tcp_iCommStatus = 0 THEN
    Tcp_xTimeout := TRUE;
    Tcp_xConnected := FALSE;
    Tcp_xOnline := FALSE;
    IF tonHb.Q THEN Tcp_iCommStatus := 4; END_IF;
    Tcp_xJogXPos := FALSE; Tcp_xJogXNeg := FALSE;
    Tcp_xSpinLeft := FALSE; Tcp_xSpinRight := FALSE;
    Tcp_xJogYPos := FALSE; Tcp_xJogYNeg := FALSE;
    Tcp_xJogZPos := FALSE; Tcp_xJogZNeg := FALSE;
    Tcp_xJogRPos := FALSE; Tcp_xJogRNeg := FALSE;
    Tcp_xHomeY := FALSE; Tcp_xHomeZ := FALSE; Tcp_xHomeR := FALSE;
    Tcp_xHomeExec := FALSE;
    Tcp_xStart := FALSE; Tcp_xEnable := FALSE;
    Tcp_xAutoStart := FALSE;
    Tcp_xForceTare := FALSE; Tcp_xForceUntare := FALSE; Tcp_xForceGuide := FALSE;
    Tcp_xForcePeakReset := FALSE;
    Tcp_xStop := TRUE;
    Tcp_xAutoAbort := TRUE;
    Tcp_xEStop := TRUE;
ELSE
    Tcp_xTimeout := FALSE;
    Tcp_xConnected := TRUE;
    Tcp_xOnline := TRUE;
END_IF;

(* ===== 状态快照编码 ===== *)
Tcp_wStatusSeq := Tcp_wStatusSeq + 1;
MB_StatusOut[0] := 19533;
MB_StatusOut[1] := 256;
MB_StatusOut[2] := Tcp_wStatusSeq;
MB_StatusOut[3] := Tcp_wLastSeq;
MB_StatusOut[4] := Tcp_wLastHb;
FOR i := 5 TO 94 DO MB_StatusOut[i] := 0; END_FOR;
MB_StatusOut[5] := INT_TO_WORD(Tcp_iCommStatus);
MB_StatusOut[6] := INT_TO_WORD(HMI_eDevState);
MB_StatusOut[7] := INT_TO_WORD(HMI_eOpMode);
MB_StatusOut[8] := INT_TO_WORD(HMI_iAlarmShow);
MB_StatusOut[9] := INT_TO_WORD(HMI_iAutoStepShow);
IF HMI_xDevStop THEN MB_StatusOut[10] := MB_StatusOut[10] OR 1; END_IF;
IF HMI_xDevRun THEN MB_StatusOut[10] := MB_StatusOut[10] OR 2; END_IF;
IF HMI_xDevError THEN MB_StatusOut[10] := MB_StatusOut[10] OR 4; END_IF;
IF HMI_xLampEStop THEN MB_StatusOut[10] := MB_StatusOut[10] OR 8; END_IF;
IF HMI_xLampEnableOk THEN MB_StatusOut[10] := MB_StatusOut[10] OR 16; END_IF;
IF HMI_xLampFault THEN MB_StatusOut[10] := MB_StatusOut[10] OR 32; END_IF;
IF HMI_xAutoBusy THEN MB_StatusOut[10] := MB_StatusOut[10] OR 64; END_IF;
IF HMI_xAutoDone THEN MB_StatusOut[10] := MB_StatusOut[10] OR 128; END_IF;
IF HMI_xHomedY THEN MB_StatusOut[10] := MB_StatusOut[10] OR 256; END_IF;
IF HMI_xHomedZ THEN MB_StatusOut[10] := MB_StatusOut[10] OR 512; END_IF;
IF HMI_xHomedR THEN MB_StatusOut[10] := MB_StatusOut[10] OR 1024; END_IF;
IF HMI_xHomeBusyY THEN MB_StatusOut[10] := MB_StatusOut[10] OR 2048; END_IF;
IF HMI_xHomeBusyZ THEN MB_StatusOut[10] := MB_StatusOut[10] OR 4096; END_IF;
IF HMI_xHomeBusyR THEN MB_StatusOut[10] := MB_StatusOut[10] OR 8192; END_IF;
IF Tcp_xConnected THEN MB_StatusOut[10] := MB_StatusOut[10] OR 16384; END_IF;
IF Tcp_xTimeout THEN MB_StatusOut[10] := MB_StatusOut[10] OR 32768; END_IF;
IF Force_xCommOk THEN MB_StatusOut[11] := MB_StatusOut[11] OR 1; END_IF;
IF Force_xTimeout THEN MB_StatusOut[11] := MB_StatusOut[11] OR 2; END_IF;
IF Force_xSlaveFail THEN MB_StatusOut[11] := MB_StatusOut[11] OR 4; END_IF;
IF Force_xTareBusy THEN MB_StatusOut[11] := MB_StatusOut[11] OR 8; END_IF;
IF Force_xTareDone THEN MB_StatusOut[11] := MB_StatusOut[11] OR 16; END_IF;
IF AxisFb_xReady THEN MB_StatusOut[11] := MB_StatusOut[11] OR 32; END_IF;
IF AxisFb_xMoveDoneX THEN MB_StatusOut[11] := MB_StatusOut[11] OR 64; END_IF;
IF AxisFb_xMoveDoneY THEN MB_StatusOut[11] := MB_StatusOut[11] OR 128; END_IF;
IF AxisFb_xFaultM1 THEN MB_StatusOut[11] := MB_StatusOut[11] OR 256; END_IF;
IF AxisFb_xFaultM2 THEN MB_StatusOut[11] := MB_StatusOut[11] OR 512; END_IF;
IF AxisFb_xFaultY THEN MB_StatusOut[11] := MB_StatusOut[11] OR 1024; END_IF;
IF AxisFb_xFaultZ THEN MB_StatusOut[11] := MB_StatusOut[11] OR 2048; END_IF;
IF AxisFb_xFaultR THEN MB_StatusOut[11] := MB_StatusOut[11] OR 4096; END_IF;
IF AxisFb_xHomedY THEN MB_StatusOut[11] := MB_StatusOut[11] OR 8192; END_IF;
IF AxisFb_xHomedZ THEN MB_StatusOut[11] := MB_StatusOut[11] OR 16384; END_IF;
IF AxisFb_xHomedR THEN MB_StatusOut[11] := MB_StatusOut[11] OR 32768; END_IF;
diTmp := REAL_TO_DINT(HMI_rForceShow * 100.0);
dwTmp := DINT_TO_DWORD(diTmp);
MB_StatusOut[12] := DWORD_TO_WORD(SHR(dwTmp, 16));
MB_StatusOut[13] := DWORD_TO_WORD(dwTmp AND 16#FFFF);
diTmp := REAL_TO_DINT(AxisFb_rPosM1 * 1000.0);
dwTmp := DINT_TO_DWORD(diTmp);
MB_StatusOut[14] := DWORD_TO_WORD(SHR(dwTmp, 16));
MB_StatusOut[15] := DWORD_TO_WORD(dwTmp AND 16#FFFF);
diTmp := REAL_TO_DINT(AxisFb_rPosM2 * 1000.0);
dwTmp := DINT_TO_DWORD(diTmp);
MB_StatusOut[16] := DWORD_TO_WORD(SHR(dwTmp, 16));
MB_StatusOut[17] := DWORD_TO_WORD(dwTmp AND 16#FFFF);
diTmp := REAL_TO_DINT(AxisFb_rPosY * 1000.0);
dwTmp := DINT_TO_DWORD(diTmp);
MB_StatusOut[18] := DWORD_TO_WORD(SHR(dwTmp, 16));
MB_StatusOut[19] := DWORD_TO_WORD(dwTmp AND 16#FFFF);
diTmp := REAL_TO_DINT(AxisFb_rPosZ * 1000.0);
dwTmp := DINT_TO_DWORD(diTmp);
MB_StatusOut[20] := DWORD_TO_WORD(SHR(dwTmp, 16));
MB_StatusOut[21] := DWORD_TO_WORD(dwTmp AND 16#FFFF);
diTmp := REAL_TO_DINT(AxisFb_rPosR * 1000.0);
dwTmp := DINT_TO_DWORD(diTmp);
MB_StatusOut[22] := DWORD_TO_WORD(SHR(dwTmp, 16));
MB_StatusOut[23] := DWORD_TO_WORD(dwTmp AND 16#FFFF);
diTmp := REAL_TO_DINT(AxisFb_rVelCmdM1 * 1000.0);
dwTmp := DINT_TO_DWORD(diTmp);
MB_StatusOut[24] := DWORD_TO_WORD(SHR(dwTmp, 16));
MB_StatusOut[25] := DWORD_TO_WORD(dwTmp AND 16#FFFF);
diTmp := REAL_TO_DINT(AxisFb_rVelCmdM2 * 1000.0);
dwTmp := DINT_TO_DWORD(diTmp);
MB_StatusOut[26] := DWORD_TO_WORD(SHR(dwTmp, 16));
MB_StatusOut[27] := DWORD_TO_WORD(dwTmp AND 16#FFFF);
(* 0.60 X 直控状态 word28..31（word5..62 每周期已清零） *)
MB_StatusOut[28] := 0;
IF Direct_xActive THEN MB_StatusOut[28] := MB_StatusOut[28] OR 1; END_IF;
IF Direct_xOnline THEN MB_StatusOut[28] := MB_StatusOut[28] OR 2; END_IF;
IF Direct_xEnable THEN MB_StatusOut[28] := MB_StatusOut[28] OR 4; END_IF;
MB_StatusOut[29] := INT_TO_WORD(REAL_TO_INT(Direct_rVelM1Act * 1000.0));
MB_StatusOut[30] := INT_TO_WORD(REAL_TO_INT(Direct_rVelM2Act * 1000.0));
MB_StatusOut[31] := Direct_wSeqEcho;
(* 0.63 X 双电机实际速度通用透传 word32..38（word5..62 每周期已清零） *)
diTmp := REAL_TO_DINT(AxisFb_rVelActM1 * 1000.0);
dwTmp := DINT_TO_DWORD(diTmp);
MB_StatusOut[32] := DWORD_TO_WORD(SHR(dwTmp, 16));
MB_StatusOut[33] := DWORD_TO_WORD(dwTmp AND 16#FFFF);
diTmp := REAL_TO_DINT(AxisFb_rVelActM2 * 1000.0);
dwTmp := DINT_TO_DWORD(diTmp);
MB_StatusOut[34] := DWORD_TO_WORD(SHR(dwTmp, 16));
MB_StatusOut[35] := DWORD_TO_WORD(dwTmp AND 16#FFFF);
MB_StatusOut[36] := 0;
IF AxisFb_xMovingM1 THEN MB_StatusOut[36] := MB_StatusOut[36] OR 1; END_IF;
IF AxisFb_xMovingM2 THEN MB_StatusOut[36] := MB_StatusOut[36] OR 2; END_IF;
IF AxisFb_xPoweredM1 THEN MB_StatusOut[36] := MB_StatusOut[36] OR 4; END_IF;
IF AxisFb_xPoweredM2 THEN MB_StatusOut[36] := MB_StatusOut[36] OR 8; END_IF;
IF AxisFb_xSyncWarn THEN MB_StatusOut[36] := MB_StatusOut[36] OR 16; END_IF;
IF AxisFb_xSyncFault THEN MB_StatusOut[36] := MB_StatusOut[36] OR 32; END_IF;
diTmp := REAL_TO_DINT(AxisFb_rSyncErr * 1000.0);
dwTmp := DINT_TO_DWORD(diTmp);
MB_StatusOut[37] := DWORD_TO_WORD(SHR(dwTmp, 16));
MB_StatusOut[38] := DWORD_TO_WORD(dwTmp AND 16#FFFF);
(* 0.68 全轴直控状态 word39..45（word5..94 每周期已清零） *)
MB_StatusOut[39] := INT_TO_WORD(REAL_TO_INT(AxisFb_rVelActY * 1000.0));
MB_StatusOut[40] := INT_TO_WORD(REAL_TO_INT(AxisFb_rVelActZ * 1000.0));
MB_StatusOut[41] := INT_TO_WORD(REAL_TO_INT(AxisFb_rVelActR * 1000.0));
MB_StatusOut[42] := 0;
IF Direct2_xActiveX THEN MB_StatusOut[42] := MB_StatusOut[42] OR 1; END_IF;
IF Direct2_xActiveY THEN MB_StatusOut[42] := MB_StatusOut[42] OR 2; END_IF;
IF Direct2_xActiveZ THEN MB_StatusOut[42] := MB_StatusOut[42] OR 4; END_IF;
IF Direct2_xActiveR THEN MB_StatusOut[42] := MB_StatusOut[42] OR 8; END_IF;
IF Direct2_xOnline THEN MB_StatusOut[42] := MB_StatusOut[42] OR 16; END_IF;
IF Direct2_xSafe THEN MB_StatusOut[42] := MB_StatusOut[42] OR 32; END_IF;
MB_StatusOut[43] := Direct2_wSeqEcho;
diTmp := REAL_TO_DINT(HMI_rForceSetEcho * 100.0);
dwTmp := DINT_TO_DWORD(diTmp);
MB_StatusOut[44] := DWORD_TO_WORD(SHR(dwTmp, 16));
MB_StatusOut[45] := DWORD_TO_WORD(dwTmp AND 16#FFFF);
(* 力峰值（SCALED_DINT ×100，高字在前）与原始计数：word46/47、word48 *)
Tcp_rForcePeak := Force_rPeak;
Tcp_wForceRaw := Force_wRaw;
diTmp := REAL_TO_DINT(Force_rPeak * 100.0);
dwTmp := DINT_TO_DWORD(diTmp);
MB_StatusOut[46] := DWORD_TO_WORD(SHR(dwTmp, 16));
MB_StatusOut[47] := DWORD_TO_WORD(dwTmp AND 16#FFFF);
MB_StatusOut[48] := Force_wRaw;
(* 0.71 M1/M2 转矩/电流（CoE 0x6077/0x6078 慢速读取，‰额定转矩/电流）word49..52；读错误 word53 bit0 *)
MB_StatusOut[49] := INT_TO_WORD(REAL_TO_INT(AxisFb_rTorqueM1));
MB_StatusOut[50] := INT_TO_WORD(REAL_TO_INT(AxisFb_rTorqueM2));
MB_StatusOut[51] := INT_TO_WORD(REAL_TO_INT(AxisFb_rCurrentM1));
MB_StatusOut[52] := INT_TO_WORD(REAL_TO_INT(AxisFb_rCurrentM2));
MB_StatusOut[53] := 0;
IF AxisFb_xParamErr THEN MB_StatusOut[53] := MB_StatusOut[53] OR 1; END_IF;
(* 0.72 驱动诊断 word54..63：M1/M2 状态字/错误码/最大转矩/正反限幅（原始 16 位） *)
MB_StatusOut[54] := AxisFb_wSwM1;
MB_StatusOut[55] := AxisFb_wErrM1;
MB_StatusOut[56] := AxisFb_wTqMaxM1;
MB_StatusOut[57] := AxisFb_wLimPM1;
MB_StatusOut[58] := AxisFb_wLimNM1;
MB_StatusOut[59] := AxisFb_wSwM2;
MB_StatusOut[60] := AxisFb_wErrM2;
MB_StatusOut[61] := AxisFb_wTqMaxM2;
MB_StatusOut[62] := AxisFb_wLimPM2;
MB_StatusOut[63] := AxisFb_wLimNM2;
(* 0.73 MDX 模式与转矩限值 word64..73 *)
MB_StatusOut[64] := AxisFb_wModeM1;
MB_StatusOut[65] := AxisFb_wTq03M1;
MB_StatusOut[66] := AxisFb_wTq04M1;
MB_StatusOut[67] := AxisFb_wTq05M1;
MB_StatusOut[68] := AxisFb_wTq06M1;
MB_StatusOut[69] := AxisFb_wModeM2;
MB_StatusOut[70] := AxisFb_wTq03M2;
MB_StatusOut[71] := AxisFb_wTq04M2;
MB_StatusOut[72] := AxisFb_wTq05M2;
MB_StatusOut[73] := AxisFb_wTq06M2;
(* 0.79 CSV 模式诊断 word74：bit0 M1 6060=9 / bit2 M2 6060=9（模式由从站 RxPDO 组态决定，只读） *)
MB_StatusOut[74] := 0;
IF AxisFb_xModeCsvM1 THEN MB_StatusOut[74] := MB_StatusOut[74] OR 1; END_IF;
IF AxisFb_xModeCsvM2 THEN MB_StatusOut[74] := MB_StatusOut[74] OR 4; END_IF;
MB_StatusOut[95] := Tcp_wStatusSeq;

(* ===== 控制源仲裁 ===== *)
xPanelOp := StartBtn OR StopBtn OR ResetBtn OR JogFwd OR JogBwd OR JogLeft OR JogRight
    OR JogUp OR JogDown OR JogClockAdd OR JogClockMis;
xTcpOp := Tcp_xOnline AND (
    Tcp_xStart OR Tcp_xStop OR Tcp_xStopHold3s OR Tcp_xAutoStart OR Tcp_xAutoAbort
    OR Tcp_xJogXPos OR Tcp_xJogXNeg OR Tcp_xSpinLeft OR Tcp_xSpinRight
    OR Tcp_xJogYPos OR Tcp_xJogYNeg OR Tcp_xJogZPos OR Tcp_xJogZNeg
    OR Tcp_xJogRPos OR Tcp_xJogRNeg
    OR Tcp_xHomeY OR Tcp_xHomeZ OR Tcp_xHomeR OR Tcp_xHomeExec
    OR Tcp_xForceGuide OR Tcp_xForceTare OR Tcp_xForceUntare);
IF NOT Tcp_xOnline THEN
    eCtrlSrc := 0;
ELSIF xTcpOp THEN
    eCtrlSrc := 1;
ELSIF xPanelOp THEN
    eCtrlSrc := 0;
END_IF;

(* 力峰值复位是显示动作，不进控制源仲裁：只要远程在线即可，避免短暂抢走 eCtrlSrc *)
HMI_xForcePeakReset := Tcp_xOnline AND Tcp_xForcePeakReset;

IF eCtrlSrc = 1 THEN
    HMI_xAutoMode := Tcp_xAutoMode;
    HMI_xJogXPos := Tcp_xJogXPos;   HMI_xJogXNeg := Tcp_xJogXNeg;
    HMI_xSpinLeft := Tcp_xSpinLeft; HMI_xSpinRight := Tcp_xSpinRight;
    HMI_xJogYPos := Tcp_xJogYPos;   HMI_xJogYNeg := Tcp_xJogYNeg;
    HMI_xJogZPos := Tcp_xJogZPos;   HMI_xJogZNeg := Tcp_xJogZNeg;
    HMI_xJogRPos := Tcp_xJogRPos;   HMI_xJogRNeg := Tcp_xJogRNeg;
    HMI_xHomeY := Tcp_xHomeY; HMI_xHomeZ := Tcp_xHomeZ; HMI_xHomeR := Tcp_xHomeR;
    HMI_iHomeAxis := Tcp_iHomeAxis; HMI_xHomeExec := Tcp_xHomeExec;
    HMI_xForceGuide := Tcp_xForceGuide;
    HMI_xForceTare := Tcp_xForceTare; HMI_xForceUntare := Tcp_xForceUntare;
    HMI_xForceSimEnable := Tcp_xForceSimEnable;
    HMI_rJogVelX := Tcp_rJogVelX; HMI_rSpinVel := Tcp_rSpinVel;
    HMI_rJogVelY := Tcp_rJogVelY; HMI_rJogVelZ := Tcp_rJogVelZ; HMI_rJogVelR := Tcp_rJogVelR;
    HMI_rAutoDistX := Tcp_rAutoDistX; HMI_rAutoVelX := Tcp_rAutoVelX;
    HMI_rAutoVelY := Tcp_rAutoVelY; HMI_rAutoVelZ := Tcp_rAutoVelZ;
    HMI_rWheelBase := Tcp_rWheelBase; HMI_rForceSet := Tcp_rForceSet;
    HMI_rForceSim := Tcp_rForceSim;
    HMI_iAutoPasses := Tcp_iAutoPasses;
    HMI_rHeadingErr := Tcp_rHeadingErr;
    HMI_rKpTrack := Tcp_rKpTrack;
    HMI_rKpForce := Tcp_rKpForce;
    HMI_rAccX := Tcp_rAccX; HMI_rDecX := Tcp_rDecX;
    HMI_rAccY := Tcp_rAccY; HMI_rDecY := Tcp_rDecY;
    HMI_rAccZ := Tcp_rAccZ; HMI_rDecZ := Tcp_rDecZ;
    HMI_rAccR := Tcp_rAccR; HMI_rDecR := Tcp_rDecR;
END_IF;

HMI_xEStop := EStop AND Tcp_xEStop AND HMI_xEStopReq;
HMI_xStart := StartBtn OR HMI_xStartReq OR (Tcp_xOnline AND Tcp_xStart);
HMI_xEnable := HMI_xStart;
HMI_xStop := StopBtn OR HMI_xStopReq OR (Tcp_xOnline AND Tcp_xStop);
HMI_xStopHold3s := ResetBtn OR HMI_xResetReq OR (Tcp_xOnline AND Tcp_xStopHold3s);
HMI_xAutoStart := (Tcp_xOnline AND Tcp_xAutoStart) OR ((eCtrlSrc = 0) AND HMI_xAutoStartReq);
HMI_xAutoAbort := HMI_xAutoAbortReq OR (Tcp_xOnline AND Tcp_xAutoAbort);
